# B&R Automation Studio project Soiled_PLC (part 15)

#### lpn.st - Implementation code
```iecst
(********************************************************************
 * COPYRIGHT --
 ********************************************************************
 * Program: pr
 * File: pr.st
 * Author: treamsbottom
 * Created: July 16, 2015
 ********************************************************************
 * Implementation of program pr
 ********************************************************************)
//V1.00.1 First Release
PROGRAM _INIT
//Configuration
mySeq						:= 31;	//Sequence number
myIO						:= 114;
myZone						:= 1;

myBag						:= 0; //Buffer Bag
myBuffBag					:= 0;

mySelectedLU_reg			:= mySeq; // D register to store selected loaded unit

bufferSettleTime			:= 300;

alarm						ACCESS ADR(Alarm[mySeq]);
bag							ACCESS ADR(Bag[myBag]);
//bag_buff					ACCESS ADR(Bag[myBuffBag]);

END_PROGRAM

PROGRAM _CYCLIC
//Inputs
i_bagAtBuffer				:= RequestRel.PN[1];//X[myIO].X01;

i_bagArriveLu[1]			:= X[myIO].X01;
i_bagArriveLu[2]			:= X[myIO].X02;

i_bagInRotaryPoint_front[1]	:= X[myIO].X03;
i_bagInRotaryPoint_rear[1]	:= X[myIO].X04;

i_bagInRotaryPoint_front[2]	:= X[myIO].X05;
i_bagInRotaryPoint_rear[2]	:= X[myIO].X06;

//Create the q for which loading unit to send to.
// N.B These input conditions are used to arrive the bag.
luWaitingLongest.input[1] := Request.LU[1]; //Loading unit does not have an empty bag space
luWaitingLongest.input[2] := NOT X[23].X01 AND NOT X[23].X02 AND NOT Y[23].Y05 AND NOT Y[23].Y06; //Loading unit 2 buffer.
luWaitingLongest.settleTime := 10;
luWaitingLongest();

o_openBuffer			:= FALSE;
o_straight				:= FALSE; // select all straight rails

FOR n := 0 TO MAX_LOADING_UNITS DO
	o_openFrontStop[n] 	:= FALSE;
	o_openRearStop[n] 	:= FALSE;
	o_rotate[n] 		:= FALSE;
END_FOR;

IF (myBag = 0) THEN
	alarm.Bag	:= mySeq + 10000;
ELSE
	alarm.Bag	:= myBag;
END_IF;

alarm.Name 		:= 0;
alarm.Beacon	:= TRUE;
alarm.Extra		:= 0;
alarm.Time		:= 3000;

//Setup Sequence
step := D[900 + mySeq];
//Setup Pulse contact
pls := (step <> lastStep);
lastStep := step;

//Sequence
IF (step = 0) THEN
	//Disabled
END_IF;

//Step 1 reset points & switch check
ton_10ms_reset(IN:=((step = 1) AND NOT Std.HaltSysZone[myZone]), PT:= 400);
IF (step = 1) THEN
	switchCheck := TRUE;
	FOR n := 1 TO MAX_LOADING_UNITS DO
		IF (i_bagArriveLu[n] OR i_bagInRotaryPoint_front[n] OR i_bagInRotaryPoint_rear[n]) THEN
			switchCheck := FALSE;
			EXIT;
		END_IF;
	END_FOR;

	o_straight := NOT Std.HaltSysZone[myZone];
	IF ton_10ms_reset.Q AND switchCheck THEN
		D[900 + mySeq] := 2;
		Count[mySeq] := Count[mySeq] + 1;
	ELSIF NOT switchCheck THEN
		alarm.Name := ALM_SWITCH_FAULT;
		alarm.Time := 0;
	END_IF;
END_IF;

ton_10ms_SettledBuffer(IN:= i_bagAtBuffer,PT:= bufferSettleTime);
//Wait for at bag buffer and  decide where to send bag
IF (step = 2) THEN
	 bagWaiting := (ton_10ms_SettledBuffer.Q AND ((bag.Cat > 0) OR(myBag = 0)));
	IF bagWaiting AND (luWaitingLongest.waitingLongest > 0)  AND NOT Std.HaltSysZone[myZone] THEN
		D[mySelectedLU_reg] := luWaitingLongest.waitingLongest; // Store the selected loaded unit to a D register so we won;t lose it
		D[900 + mySeq] := 3;
	END_IF;
	IF (myBag > 0) AND ton_10ms_SettledBuffer.Q  AND (bag.Cat = 0) THEN
		alarm.Name := ALM_BAG_DATA_ERROR;
	END_IF;
END_IF;

loadingUnit := D[mySelectedLU_reg];
//open buffer and wait for trolley past stop
releaseValid := (loadingUnit > 0);
IF (step = 3) THEN
	//o_straight := 1;
	o_openBuffer := releaseValid;
	FOR n := loadingUnit TO 1 BY -1 DO;
		o_openFrontStop[n] := 1;	// Open all front stops up to and including the selected unit;
		o_openRearStop[n-1] := 1;	// Open all rear stops up to the selected unitl
	END_FOR;
	IF i_bagInRotaryPoint_rear[loadingUnit] OR i_bagArriveLu[loadingUnit] THEN //i_bagArriveLu[loadingUnit]
		D[900 + mySeq] := 4;
	END_IF;
	IF releaseValid  AND NOT Std.HaltSysZone[myZone] THEN
		alarm.Name := ALM_BAG_NOT_ARRIVED;
	END_IF;
END_IF;

//bag settles in rotary points.
ton_SettledInPoint(IN:= (i_bagInRotaryPoint_front[loadingUnit] AND i_bagInRotaryPoint_rear[loadingUnit]), PT := 300);
IF (step = 4) THEN
	//o_straight := 1;
	FOR n := loadingUnit TO 1 BY -1 DO;
		o_openFrontStop[n-1] := 1;	// Open all rear stops up to the selected unitl
		o_openRearStop[n-1] := 1;	// Open all rear stops up to the selected unitl
	END_FOR;
	IF ton_SettledInPoint.Q   AND NOT Std.HaltSysZone[myZone] THEN
		D[900 + mySeq] := 5;
	ELSIF NOT Std.HaltSysZone[myZone] THEN
		alarm.Name := ALM_BAG_NOT_SETTLED;
	END_IF;
END_IF;

//rotate points
ton_rotatePoints(IN:= (step = 5),PT:= 400);
IF (step = 5) THEN
	o_rotate[loadingUnit] := 1;
	IF ton_rotatePoints.Q AND NOT Std.HaltSysZone[myZone] THEN
		D[900 + mySeq] := 6;
	END_IF;
END_IF;

//release bag
IF (step = 6) THEN
	o_rotate[loadingUnit] := 1;
	o_openFrontStop[loadingUnit] := luWaitingLongest.input[loadingUnit];
	o_openRearStop[loadingUnit] := luWaitingLongest.input[loadingUnit];
	IF NOT luWaitingLongest.input[loadingUnit] THEN
		D[900 + mySeq] := 1;
	END_IF;
	alarm.Name := ALM_BAG_NOT_RELEASED;
END_IF;

//-----------------------------------
//PLC Outputs - adjust TO suit system
//-----------------------------------

//Y[myIO].Y05 := o_openBuffer;
EnableRel.PN[1]		:= o_openBuffer;

Y[380].Y01	:= o_straight;
Y[380].Y02  := o_rotate[1];
Y[380].Y03	:= o_straight;
Y[380].Y04  := o_rotate[1];
Y[380].Y05  := o_openFrontStop[1];
Y[380].Y06  := o_openRearStop[1];

Y[382].Y01	:= o_straight;
Y[382].Y02  := o_rotate[2];
Y[382].Y03	:= o_straight;
Y[382].Y04  := o_rotate[2];
Y[382].Y05  := o_openFrontStop[2];
Y[382].Y06  := o_openRearStop[2];

//Alarms
timerAlarm(IN := NOT pls AND (alarm.Name > 0),PT:= alarm.Time);

alarm.On 	:= timerAlarm.Q;
alarm.ET 	:= timerAlarm.ET;

END_PROGRAM
```

#### lpn.var - Local variables
```iecst
(********************************************************************
 * COPYRIGHT --
 ********************************************************************
 * Program: pr
 * File: pr.var
 * Author: treamsbottom
 * Created: July 16, 2015
 ********************************************************************
 * Local variables of program pr
 ********************************************************************)
VAR CONSTANT
	MAX_LOADING_UNITS : USINT := 2;
END_VAR
VAR
	mySeq : UINT;
	myIO : UINT;
	myZone : UINT;
	myBag : UINT;
	i_bagAtBuffer : BOOL;
	o_openBuffer : BOOL;
	step : UINT;
	pls : BOOL;
	timerAlarm : TON_10ms;
END_VAR
VAR RETAIN
	lastStep : UINT;
END_VAR
VAR
	bufferSettleTime : UDINT;
	myOutBag : UINT;
	myBuffBag : UINT;
	myCan : UINT;
	alarm : REFERENCE TO Alm;
	bag : REFERENCE TO Bag_typ;
	bag_buff : REFERENCE TO Bag_typ;
	bag_out : REFERENCE TO Bag_typ;
	can : REFERENCE TO CAN_Vars;
	ton_10ms_reset : TON_10ms := (0);
	bagWaiting : BOOL := 0;
	ton_10ms_SettledBuffer : TON_10ms := (0);
	luWaitingLongest : getWaitingLongest := (0);
	mySelectedLU_reg : UINT := 0;
	loadingUnit : UINT := 0;
	releaseValid : BOOL := 0;
	o_openFrontStop : ARRAY[0..MAX_LOADING_UNITS] OF BOOL := [0];
	o_openRearStop : ARRAY[0..MAX_LOADING_UNITS] OF BOOL := [0];
	i_bagArriveLu : ARRAY[0..MAX_LOADING_UNITS] OF BOOL := [0];
	o_rotate : ARRAY[0..MAX_LOADING_UNITS] OF BOOL := [0];
	o_straight : BOOL := FALSE;
	i_bagInRotaryPoint_front : ARRAY[0..MAX_LOADING_UNITS] OF BOOL := [0];
	i_bagInRotaryPoint_rear : ARRAY[0..MAX_LOADING_UNITS] OF BOOL := [0];
	ton_SettledInPoint : TON_10ms := (0);
	ton_rotatePoints : TON_10ms := (0);
	switchCheck : BOOL := 0;
	n : UINT := 0;
END_VAR
```

### Program Logical/BaseStandards/TwinRailLoadingUnit/lpf (IEC, version 1.00.1) - *Twin rail loading offgoing

#### lpf.st - Implementation code
```iecst
(********************************************************************
 * COPYRIGHT --
 ********************************************************************
 * Program: pr
 * File: pr.st
 * Author: treamsbottom
 * Created: July 16, 2015
 ********************************************************************
 * Implementation of program pr
 ********************************************************************)
//V1.00.1 First Release
PROGRAM _INIT
//Configuration
mySeq						:= 32;	//Sequence number
myIO						:= 115;	// IO for switches
myZone						:= 1;
myPF						:= 1;

myBag						:= 207; //transit Bag
myRelLine					:= 0; // Release Line - Set to 0 to Request Release

myLuBag[1]					:= 203;
myLuBag[2]					:= 201;

mySelectedLU_reg			:= mySeq; // D register to store selected loaded unit
bufferSettleTime			:= 300;

myOutBag					:= Line[myRelLine].LastBag;

alarm						ACCESS ADR(Alarm[mySeq]);
bag							ACCESS ADR(Bag[myBag]);
bag_out						ACCESS ADR(Bag[myOutBag]);
line_release				ACCESS ADR(Line[myRelLine]);

END_PROGRAM

PROGRAM _CYCLIC
//Inputs

i_bagInRotaryPoint_front[1]	:= X[myIO].X03;
i_bagInRotaryPoint_rear[1]	:= X[myIO].X04;

i_bagInRotaryPoint_front[2]	:= X[myIO].X05;
i_bagInRotaryPoint_rear[2]	:= X[myIO].X06;

i_bagAtBufferOut 		:= FALSE; // Any Single bag buffer out IO.
i_bufferOutOpen			:= FALSE;

//Create the q for which loading unit to send to.
// N.B These input conditions are used to arrive the bag.
luWaitingLongest.input[1] := X[21].X03 AND X[21].X04 AND (Bag[myLuBag[1]].Cat > 0); //Loading unit does not have an full bag space
luWaitingLongest.input[2] := RequestRel.LU[2];
luWaitingLongest.settleTime := bufferSettleTime;
luWaitingLongest();

o_straight				:= FALSE; // select all straight rails
Request.PF[myPF]		:= FALSE;
RequestRel.PF[myPF]		:= FALSE;

FOR n := 0 TO MAX_LOADING_UNITS DO
	o_openStops[n]		:= FALSE;	// Stop on rotary points.
	o_rotate[n] 		:= FALSE;
	o_release[n]		:= FALSE;	// Release from loading unit or buffer.
END_FOR;

IF (myBag = 0) THEN
	alarm.Bag	:= mySeq + 10000;
ELSE
	alarm.Bag	:= myBag;
END_IF;

alarm.Name 		:= 0;
alarm.Beacon	:= TRUE;
alarm.Extra		:= 0;
alarm.Time		:= 3000;

//Setup Sequence
step := D[900 + mySeq];
//Setup Pulse contact
pls := (step <> lastStep);
lastStep := step;

//Sequence
IF (step = 0) THEN
	//Disabled
END_IF;

//Step 1 reset points & switch check
ton_10ms_reset(IN:=((step = 1) AND NOT Std.HaltSysZone[myZone]), PT:= 400);
IF (step = 1) THEN
	switchCheck := TRUE;
	FOR n := 1 TO MAX_LOADING_UNITS DO
		IF (i_bagInRotaryPoint_front[n] OR i_bagInRotaryPoint_rear[n]) THEN
			switchCheck := FALSE;
			EXIT;
		END_IF;
	END_FOR;
	o_straight := NOT Std.HaltSysZone[myZone];
	IF ton_10ms_reset.Q AND switchCheck AND (bag.Cat = 0) THEN
		D[900 + mySeq] := 2;
		Count[mySeq] := Count[mySeq] + 1;
	ELSIF NOT switchCheck THEN
		alarm.Name := ALM_SWITCH_FAULT;
		alarm.Time := 0;
	ELSIF (bag.Cat > 0) THEN
		alarm.Name := ALM_BAG_DATA_ERROR;
		alarm.Time := 0;
	END_IF;
END_IF;

//Wait for at bag buffer and  decide where to send bag
IF (step = 2) THEN
	releaseOk := (bag.Cat = 0);// We don;t have to check the loading unit bag data.. the queue is already checking it,
	IF releaseOk AND (luWaitingLongest.waitingLongest > 0)  AND NOT Std.HaltSysZone[myZone] THEN
		D[mySelectedLU_reg] := luWaitingLongest.waitingLongest; // Store the selected loaded unit to a D register so we won;t lose it
		D[900 + mySeq] := 3;
	ELSIF NOT releaseOk  AND NOT Std.HaltSysZone[myZone] THEN
		alarm.Name := ALM_BAG_DATA_ERROR;
		alarm.Time := 0;
	END_IF;
END_IF;

loadingUnit := D[mySelectedLU_reg];

//rotate points
ton_rotatePoints(IN:= ((step = 3) OR (step = 5)) ,PT:= 400);
IF (step = 3) THEN
	o_rotate[loadingUnit] := 1;
	IF ton_rotatePoints.Q  AND NOT Std.HaltSysZone[myZone] THEN
		D[900 + mySeq] := 4;
	END_IF;
END_IF;

releaseOk := (bag.Cat = 0) AND (Bag[myLuBag[loadingUnit]].Cat > 0) AND NOT Std.HaltSysZone[myZone];
//bag settles in point
ton_SettledInPoint(IN:= (i_bagInRotaryPoint_front[loadingUnit] AND i_bagInRotaryPoint_rear[loadingUnit]), PT := 300);
IF (step = 4) THEN
	o_rotate[loadingUnit] := 1;
	o_release[loadingUnit] := releaseOk;
	IF ton_SettledInPoint.Q AND releaseOk  THEN
		bag := Bag[myLuBag[loadingUnit]];
		Bag[myLuBag[loadingUnit]] := Bag[0];
		D[900 + mySeq] := 5;
	ELSIF NOT releaseOk AND NOT Std.HaltSysZone[myZone] THEN
		IF (bag.Cat > 0) THEN
			alarm.Name := ALM_BAG_DATA_ERROR;
			alarm.Time := 0;
		ELSE
			alarm.Name 	:= ALM_BAG_DATA_ERROR;
			alarm.Time 	:= 0;
			alarm.Bag 	:= myLuBag[loadingUnit];
		END_IF;
	ELSE
		alarm.Name := ALM_BAG_NOT_SETTLED;
	END_IF;
END_IF;

//rotate points back to straight
IF (step = 5) THEN
	o_straight	:= 1;
	IF ton_rotatePoints.Q AND NOT EnableRel.PF[myPF] THEN
		D[900 + mySeq] := 6;
	ELSIF EnableRel.PF[myPF] THEN
		alarm.Name := ALM_BAG_DATA_ERROR;
	END_IF;
END_IF;

//Check for line space.
IF (step = 6) THEN
	releaseValid := (NOT i_bagAtBufferOut AND NOT i_bufferOutOpen AND (bag.Cat > 0) AND (bag_out.Cat = 0));
	o_straight	:= 1;
	IF NOT Std.HaltSysZone[myZone] THEN
		IF (myRelLine > 0) THEN
			IF (line_release.Clear AND releaseValid) THEN
				C[myRelLine] := 0;
				D[900 + mySeq] := 7;
			END_IF;
			IF (line_release.Clear AND i_bagAtBufferOut) THEN
				alarm.Name := ALM_SWITCH_FAULT;
			ELSIF (bag.Cat = 0) THEN
				alarm.Name := ALM_BAG_DATA_ERROR;
				alarm.Time := 0;
			ELSIF line_release.Clear AND (bag_out.Cat > 0) THEN
				alarm.Name := ALM_BAG_DATA_ERROR;
				alarm.Bag := myOutBag;
				alarm.Time := 0;
			END_IF;
		ELSE
			RequestRel.PF[myPF] := releaseValid;
			IF EnableRel.PF[myPF] AND releaseValid THEN
				D[900 + mySeq] := 7;
			ELSIF (myBag > 0) AND (bag.Cat = 0) THEN
				alarm.Name := ALM_BAG_DATA_ERROR;
				alarm.Time := 0;
			ELSIF (myOutBag > 0) AND (bag_out.Cat > 0) THEN
				alarm.Name := ALM_BAG_DATA_ERROR;
				alarm.Bag := myOutBag;
				alarm.Time := 0;
			END_IF;
		END_IF;
	END_IF;
END_IF;

//Release bag.
IF (step = 7) THEN
	IF (NOT i_bagAtBufferOut AND NOT i_bufferOutOpen AND (bag.Cat > 0) AND (bag_out.Cat = 0) AND NOT Std.HaltSysZone[myZone]) THEN
		releaseValid := 1;
	END_IF;
	FOR n := loadingUnit TO 1 BY - 1 DO
		o_openStops[n] := releaseValid;
	END_FOR;
	o_straight := 1;
	IF releaseValid THEN
		IF (myRelLine > 0) THEN
			IF line_release.Trip THEN
				bag_out := bag;
				bag := Bag[0];
				D[900 + mySeq] := 1;
			END_IF;
		ELSE
			IF NOT EnableRel.PF[myPF] AND (bag.Cat = 0) THEN // Make sure data is copied out by enabling sequence.
				D[900 + mySeq] := 1;
			ELSIF NOT EnableRel.PF[myPF] AND (bag.Cat > 0) THEN
				alarm.Name := ALM_BAG_DATA_ERROR;
			END_IF;
		END_IF;
	ELSIF i_bagAtBufferOut OR i_bufferOutOpen THEN
		alarm.Name := ALM_SWITCH_FAULT;
		alarm.Time := 0;
	ELSIF (bag.Cat = 0) THEN
		alarm.Name := ALM_BAG_DATA_ERROR;
		alarm.Time := 0;
	ELSIF (bag_out.Cat > 0) THEN
		alarm.Name := ALM_BAG_DATA_ERROR;
		alarm.Bag := myOutBag;
		alarm.Time := 0;
	END_IF;
ELSE
	releaseValid := 0;
END_IF;

//-----------------------------------
//PLC Outputs - adjust TO suit system
//-----------------------------------

Y[21].Y07 := o_release[1];
Y[21].Y08 := o_release[1];

EnableRel.LU[2] := o_release[2];

Y[381].Y01	:= o_straight;
Y[381].Y02  := o_rotate[1];
Y[381].Y03	:= o_straight;
Y[381].Y04  := o_rotate[1];
Y[381].Y05  := o_openStops[1];
Y[381].Y06  := o_openStops[1];

Y[383].Y01	:= o_straight;
Y[383].Y02  := o_rotate[2];
Y[383].Y03	:= o_straight;
Y[383].Y04  := o_rotate[2];
Y[383].Y05  := o_openStops[2];
Y[383].Y06  := o_openStops[2];

//Alarms
timerAlarm(IN := NOT pls AND (alarm.Name > 0),PT:= alarm.Time);

alarm.On 	:= timerAlarm.Q;
alarm.ET 	:= timerAlarm.ET;

END_PROGRAM
```

#### lpf.var - Local variables
```iecst
(********************************************************************
 * COPYRIGHT --
 ********************************************************************
 * Program: pr
 * File: pr.var
 * Author: treamsbottom
 * Created: July 16, 2015
 ********************************************************************
 * Local variables of program pr
 ********************************************************************)
VAR CONSTANT
	MAX_LOADING_UNITS : USINT := 2;
END_VAR
VAR
	mySeq : UINT;
	myIO : UINT;
	myZone : UINT;
	myBag : UINT;
	step : UINT;
	pls : BOOL;
	timerAlarm : TON_10ms;
END_VAR
VAR RETAIN
	lastStep : UINT;
END_VAR
VAR
	myOutBag : UINT;
	myLuBag : ARRAY[0..MAX_LOADING_UNITS] OF UINT;
	alarm : REFERENCE TO Alm;
	bag : REFERENCE TO Bag_typ;
	bag_out : REFERENCE TO Bag_typ;
	ton_10ms_reset : TON_10ms := (0);
	luWaitingLongest : getWaitingLongest := (0);
	mySelectedLU_reg : UINT := 0;
	loadingUnit : UINT := 0;
	releaseValid : BOOL := 0;
	o_openStops : ARRAY[0..MAX_LOADING_UNITS] OF BOOL := [0];
	o_rotate : ARRAY[0..MAX_LOADING_UNITS] OF BOOL := [0];
	o_straight : BOOL := FALSE;
	i_bagInRotaryPoint_front : ARRAY[0..MAX_LOADING_UNITS] OF BOOL := [0];
	i_bagInRotaryPoint_rear : ARRAY[0..MAX_LOADING_UNITS] OF BOOL := [0];
	ton_SettledInPoint : TON_10ms := (0);
	ton_rotatePoints : TON_10ms := (0);
	switchCheck : BOOL := 0;
	o_release : ARRAY[0..MAX_LOADING_UNITS] OF BOOL := [0];
	releaseOk : BOOL := FALSE;
	myRelLine : UINT := 0;
	bufferSettleTime : UINT := 0;
	line_release : REFERENCE TO Line_Typ;
	i_bagAtBufferOut : BOOL := 0;
	i_bufferOutOpen : BOOL := 0;
	myPF : UINT := 0;
	n : UINT := 0;
END_VAR
```

### Program Logical/BaseStandards/11_spi1 (IEC) - * SPI1 Pneumatic Incline Up 1

#### 11_spi1.var
```iecst
VAR RETAIN
	STEP	:UINT;
	PLS	:BOOL;
	LASTSTEP	:UINT;
	BagSettled	:BOOL;
	BagSettledET	:TIME;
	O_OpenBufferStop	:BOOL;
	BagSettledBuffer	:BOOL;
	I_BaginIncline	:BOOL;
	BagSettledBufferET	:TIME;
	I_BagAtBuffer	:BOOL;
	I_CarrAtBottom	:BOOL;
	I_CarrAtTop	:BOOL;
	O_MoveDown	:BOOL;
END_VAR

VAR
	TempDownTime	:BOOL;
	TempDownTimeET	:TIME;
END_VAR
```

#### 11_spi1Cyclic.ab
```automation-basic
PROGRAM _CYCLIC
	(* cyclic program *)

;Sequence 11 - Pneumatic Incline 1 D[911]

;Incline Conveyor

;-----------------------------------------
;Revision 1.00 17/01/2006 D.J. First Issue
;-----------------------------------------

TON_10ms(O_MoveDown,1000,TempDownTime,TempDownTimeET)

I_BagAtBuffer			= X[8].X12
I_BaginIncline			= X[8].X13
I_CarrAtBottom			= X[8].X14
I_CarrAtTop				= X[8].X15

O_MoveDown 				= FALSE
O_OpenBufferStop		= FALSE

Request.PI[1]			= FALSE

Alarm[11].Name 			= 0
Alarm[11].Bag			= 10011
Alarm[11].Beacon		= TRUE

;Setup Sequence
;--------------
STEP = D[911]
;Setup Pulse contact
PLS = (STEP <> LASTSTEP)
LASTSTEP = STEP

;Allow carriage to go up to top
IF (STEP = 1) THEN
	IF I_CarrAtTop THEN
		D[911] = 2
	ENDIF
	IF NOT Std.HaltSys THEN
		Alarm[11].Name = almCarriageMoveFault
	ENDIF
ENDIF

;Check for bag at buffer
TON_10ms(I_BagAtBuffer,300,BagSettledBuffer,BagSettledBufferET)
IF (STEP = 2) THEN
	IF BagSettledBuffer THEN
		D[911] = 3
	ENDIF
ENDIF

;Open Buffer Stop on steps 3
IF (STEP >= 3) AND (STEP <= 3) THEN
	O_OpenBufferStop = TRUE
ENDIF

;Wait for bag in incline
IF (STEP = 3) THEN
	IF I_BaginIncline THEN
		D[911] = 4
	ENDIF
;	Alarm[11].Name = almBagNotArrived
ENDIF

;Let bag settle at base of incline
TON_10ms(I_BaginIncline,300,BagSettled,BagSettledET)
IF (STEP = 4) THEN
	IF BagSettled THEN
		D[911] = 5
	ENDIF
	Alarm[11].Name = almBagNotSettled
ENDIF

;Move carriage down to bottom
IF (STEP = 5) THEN
	O_MoveDown = TRUE
	IF I_CarrAtBottom THEN
		D[911] = 6
	ENDIF
	Alarm[11].Name = almCarriageMoveFault
ENDIF

;Allow carriage to move up to top
IF (STEP = 6) THEN
	IF I_CarrAtTop THEN
		D[911] 	= 7
	ENDIF
	Alarm[11].Name = almCarriageMoveFault
ENDIF

;Wait for space at empty bag buffer
IF (STEP = 7) THEN
	Request.PI[1] = TRUE
	IF Line[18].Clear AND BagSettled THEN
		D[911] 	= 8
	ENDIF
ENDIF

;Move carriage down to bottom
IF (STEP = 8) THEN
	O_MoveDown = TRUE
	IF I_CarrAtBottom THEN
		D[911] = 9
	ENDIF
	Alarm[11].Name = almCarriageMoveFault
ENDIF

;Allow carriage to move up releasing bag
IF (STEP = 9) THEN
	IF PLS THEN
		C[18] = 0
	ENDIF
	IF Line[18].Trip THEN
		D[911] = 1
	ENDIF
	Alarm[11].Name = almBagNotReleased
ENDIF

;Alarms
TON_10ms(NOT PLS AND (Alarm[11].Name > 0),3000,Alarm[11].On,Alarm[11].ET)

Y[8].Y12 = O_OpenBufferStop
Y[8].Y13 = O_MoveDown
END_PROGRAM
```

### Program Logical/BaseStandards/41_stnsa1 (IEC) - *Sorting Stations--

#### stnsa.ab
```automation-basic
PROGRAM _CYCLIC
(* cyclic program *)

;Honeycombe Sorting Station Control
;----------------------------------------------------
;Revision 1.00 10/01/2002 D.J. First Issue
;Revision 2.00 07/02/2005 D.J. Removed Stn Mix
;Revision 3.00 22/08/2006 D.J. Changed to timer array
;----------------------------------------------------

mySeq = 34
Bank = 1

;Timers
OpenTime  = 700
CloseTime = 500

ContinuousSort = FALSE;(D[994] = 0)

;Lamp Test from TrackView
IF (BIT_TST(D[998],0) = 1) THEN
	LampTest = TRUE

ELSE
	LampTest = FALSE
ENDIF

	LOOP x = 1 TO Ldg[Bank].NoStations DO
		n = Ldg[Bank].Stations[x]

		;Parts Loads
		TimerPartLoad[n].IN		= I_PartLoad[n]
		TimerPartLoad[n].PT		= 100
		TimerPartLoad[n] FUB TON_10ms()

		IF TimerPartLoad[n].Q THEN
			D[800 + n] = 1
		ENDIF

		;Bag open timers
		TimerOpen[n].IN 		= OpenBag[n]
		TimerOpen[n].PT			= OpenTime
		TimerOpen[n] FUB TON_10ms()

		BagOpened[n] 			= TimerOpen[n].Q
		BagOpenedET[n]			= TimerOpen[n].ET

		;Bag closed timers
		TimerClosed[n].IN 		= NOT OpenBag[n]
		TimerClosed[n].PT		= CloseTime
		TimerClosed[n] FUB TON_10ms()

		BagClosed[n] 			= TimerClosed[n].Q
		BagClosedET[n]			= TimerClosed[n].ET

		;Update bag weight
		StnBag = LDG_GetBagFromStation(Std.StationBagsStart,n)
		Bag[StnBag].Wgt 		= Stn[n].Weight
		Bag[StnBag].Cnt 		= Stn[n].Count

		;Update Bag ID if cleared or zero
		IF ((BidStn > 0) AND (Bag[StnBag].Bid = 0) AND (Bag[StnBag].Cat > 0)) THEN
			Bag[StnBag].Bid = UINT(BidStn)
			BidStn			= 0
		ENDIF

		;Move bags from Display buffer position into Search array,,
		myDisplayBag = LDG_GetBagFromStation(Std.StationBagDisplay,n)

		;Keep Weight Live on Display
		Bag[myDisplayBag].Wgt = Stn[n].Weight
		Update = FALSE
		IF (Bag[StnBag].Cat <> Bag[myDisplayBag].Cat) THEN
			Update = TRUE
		ELSE IF (Bag[StnBag].Cus <> Bag[myDisplayBag].Cus) THEN
			Update = TRUE
		ELSE IF (Bag[StnBag].Prg <> Bag[myDisplayBag].Prg) THEN
			Update = TRUE
		ENDIF
		IF (Bag[myDisplayBag].Cat = Std.MaxCats) THEN
			Update = FALSE ; Do not update bag if Empty Bag is assigned.
			CloseFlap[n] = TRUE
		ELSE
			CloseFlap[n] = FALSE
		ENDIF

		;Flap close after above SP2 for 1 second
		TimerFlapClose[n].IN 	= Stn[n].SP2 AND (Bag[myDisplayBag].Cat <> Std.MaxCats)
		TimerFlapClose[n].PT	= 200 ;4 sec
		TimerFlapClose[n] FUB TON_10ms()

		IF ContinuousSort THEN
			AutoPurgeTrig[n].CLK = Update
			AutoPurgeTrig[n] FUB R_TRIG()
			IF AutoPurgeTrig[n].Q THEN
				newBag[n] = TRUE
			ENDIF

			IF (newBag[n] AND Std.AutoPurge AND NOT Stn[n].CloseFlap AND NOT Stn[n].ManualRelease AND NOT Stn[n].Purge AND NOT Stn[n].PurgeReverse)THEN
				D[800 + n] = 2 ; Bag change detected automatically purge the station... Weight is check in ZZstn
				newBag[n] = FALSE
			ENDIF

			IF ((NOT Stn[n].CloseFlap AND NOT Stn[n].ManualRelease AND NOT Stn[n].Purge AND NOT Stn[n].PurgeReverse AND (D[800 + n] = 0)) OR  (Bag[StnBag].Cat = 0)) THEN ;AND NOT Stn[n].SP2 THEN
				IF Update THEN;(Update AND (n <> 12)) THEN
					myBid = Bag[StnBag].Bid
					Bag[StnBag] = Bag[myDisplayBag]
					Bag[StnBag].Bid = myBid
				ENDIF
			ENDIF
		ELSE
			IF Update THEN
				myBid = Bag[StnBag].Bid
				Bag[StnBag] = Bag[myDisplayBag]
				Bag[StnBag].Bid = myBid
			ENDIF
		ENDIF

		;Ensure Display Bag has a  Bag ID
		IF ((BidStn > 0) AND (Bag[myDisplayBag].Bid = 0) AND  (Bag[myDisplayBag].Cat > 0)) THEN
			Bag[myDisplayBag].Bid = UINT(BidStn)
			BidStn			= 0
		ENDIF

		Alarm[mySeq + n].Name 		= 0
		Alarm[mySeq + n].Bag		= StnBag
		Alarm[mySeq + n].Beacon	= FALSE
		Alarm[mySeq + n].Extra		= 0
		Alarm[mySeq + n].Time		= 4000

		Stn[n].LampOn 		= FALSE
		Stn[n].GreenLamp	= FALSE

		STEP = D[900 + mySeq + n]
		;Setup Pulse contact
		PLS[n] = (STEP <> LASTSTEP[n])
		LASTSTEP[n] = STEP

		;Step 0 - Disabled
		IF (STEP = 0) THEN
			Stn[n].LampOn = TRUE
			Stn[n].CloseFlap = ((Bag[StnBag].Cat <> Bag[myDisplayBag].Cat))
			Stn[n].QTime = 0
			Stn[n].ManualRelease = 0
			Stn[n].Purge = 0
			;Disabled
		ENDIF

		IF (STEP = 1) THEN
			Stn[n].LampOn = TRUE
			Stn[n].GreenLamp = FALSE
			Stn[n].CloseFlap = TRUE
			myStnReg = (n > 32)
			IF (myStnReg = 0)THEN
				myStnBit =	n - 1
			ELSE IF (myStnReg = 1)THEN
				myStnBit = 	n - 33
			ELSE
				myStnBit = 0
			ENDIF
			Std.PurgeBank[Bank].StationsStatus[myStnReg] = BIT_CLR(Std.PurgeBank[Bank].StationsStatus[myStnReg],myStnBit)

	;		Stn[n].Purge = FALSE
	;		Stn[n].PurgeReverse = FALSE
			IF D[900 + Std.StationBankReg + Bank] = n THEN
				D[900 + Std.StationBankReg + Bank] = 0
			ENDIF
			IF BagClosed[n] THEN
				D[900 + mySeq + n] = 2
			ENDIF
			Alarm[mySeq + n].Name = almStationNotClosed
		ENDIF

		IF (STEP = 2) THEN
			Stn[n].LampOn = ((Stn[n].SP1 AND Std.Clock2s) OR Stn[n].SP2 OR (Stn[n].SP3 AND Std.Clock200ms))
			Stn[n].GreenLamp = ((NOT Stn[n].SP2 AND NOT Stn[n].SP3) OR TimerFlapClose[n].Q)
			;Close the flaps when the bag is above SP2
			IF TimerFlapClose[n].Q OR Stn[n].ManualRelease OR Stn[n].Purge OR Stn[n].PurgeReverse THEN
				Stn[n].CloseFlap 	= ContinuousSort
			ENDIF
			;Stop flap closing / re-open is bag below 3kg
			IF (Stn[n].Weight < 30) THEN
				Stn[n].CloseFlap 	= FALSE
			ENDIF
			IF ((D[900 + Std.StationBankReg + Bank] = n) AND Ldg[Bank].EnableStnRelease) THEN
				D[900 + mySeq + n] = 3
			ENDIF
			IF ((Bag[StnBag].Prg > 0) AND Stn[n].SP3) THEN
				Alarm[mySeq + n].Name = almBagOverWeight
			ENDIF
		ENDIF

		IF (STEP = 3) THEN
			Stn[n].LampOn = TRUE
			Stn[n].CloseFlap = ContinuousSort
			Stn[n].GreenLamp = TimerFlapClose[n].Q

			AllowRelease[n]  = TRUE

			IF (BagOpened[n] AND ((Stn[n].Weight < 30) OR Test.Stations) AND Ldg[Bank].BeltHasRun) THEN
				Stn[n].QTime 	= 0
				D[900 + mySeq + n] = 1
			ENDIF
			IF (Stn[n].Weight >= 30) THEN
				Alarm[mySeq + n].Name = almStationNotEmpty
			ENDIF
		ELSE
			AllowRelease[n]= FALSE
		ENDIF

		OpenBag[n] = AllowRelease[n];(STEP = 3)

		;Lamp Test
		IF LampTest THEN
			Stn[n].LampOn = TRUE
		ENDIF

		;Alarm timer
		TimerAlarm[n].IN 	= NOT PLS[n] AND (Alarm[mySeq + n].Name > 0)
		TimerAlarm[n].PT	= Alarm[mySeq + n].Time
		TimerAlarm[n] FUB TON_10ms()

		Alarm[mySeq + n].ET	= TimerAlarm[n].ET
		Alarm[mySeq + n].On 	= TimerAlarm[n].Q

;	Y[300 + n].Y07 = Stn[n].LampOn
;	Y[300 + n].Y05 = Stn[n].CloseFlap OR testClose
;	Y[300 + n].Y06 = Stn[n].GreenLamp
;	Y[300 + n].Y04 = OpenBag[n]

ENDLOOP

;Outputs
;-------
;	YG05 = OpenBag[1]
;	YG06 = OpenBag[2]
;	YG07 = OpenBag[3]
;	YG08 = OpenBag[4]
;	YH05 = OpenBag[5]
;	YH06 = OpenBag[6]
;	YH07 = OpenBag[7]
;	YH08 = OpenBag[8]
;	YJ05 = OpenBag[9]
;	YJ06 = OpenBag[10]
;	YJ07 = OpenBag[11]
;	YJ08 = OpenBag[12]
;	YK05 = OpenBag[13]
;	YK06 = OpenBag[14]
;	YK07 = OpenBag[15]
;	YK08 = OpenBag[16]

	Y[31].Y05 = OpenBag[1] ;ok
	Y[31].Y06 = OpenBag[2]
	Y[31].Y07 = OpenBag[3]
	Y[31].Y08 = OpenBag[4]

	Y[32].Y05 = OpenBag[5];ok
	Y[32].Y06 = OpenBag[6]
	Y[32].Y07 = OpenBag[7]
	Y[32].Y08 = OpenBag[8]

	Y[33].Y05 = OpenBag[9]
	Y[33].Y06 = OpenBag[10]
	Y[33].Y07 = OpenBag[11]
	Y[33].Y08 = OpenBag[12]

	Y[34].Y05 = OpenBag[13]
	Y[34].Y06 = OpenBag[14]
	Y[34].Y07 = OpenBag[15]
	Y[34].Y08 = OpenBag[16]

	Y[31].Y01 = Stn[1].LampOn ;ok
	Y[31].Y02 = Stn[2].LampOn
	Y[31].Y03 = Stn[3].LampOn
	Y[31].Y04 = Stn[4].LampOn

	Y[32].Y01 = Stn[5].LampOn ;ok
	Y[32].Y02 = Stn[6].LampOn
	Y[32].Y03 = Stn[7].LampOn
	Y[32].Y04 = Stn[8].LampOn

	Y[33].Y01 = Stn[9].LampOn
	Y[33].Y02 = Stn[10].LampOn
	Y[33].Y03 = Stn[11].LampOn
	Y[33].Y04 = Stn[12].LampOn

	Y[34].Y01 = Stn[13].LampOn
	Y[34].Y02 = Stn[14].LampOn
	Y[34].Y03 = Stn[15].LampOn
	Y[34].Y04 = Stn[16].LampOn

END_PROGRAM
```

### Program Logical/BaseStandards/15_cdc1 (IEC) - * SDC2 Machine 2 CAN

#### 7_sdc2Cyclic.ab
```automation-basic
PROGRAM _CYCLIC
	(* cyclic program *)

;Sequence 7 - Discharger 2 D[907]

;-----------------------------------------
;Revision 1.00 19/12/2005 D.J. First Issue
;-----------------------------------------

DischargerEnable 		= ((D[13] > 0) AND NOT Std.HaltSys)

;I_BagAtBuffer			= X[6].X07
I_OpenBag				= CAN[2].DropLoad OR TestDrop
I_LoadDropped			= CAN[2].LoadDropped OR TestDropped
I_BagAtBuffer			= X[6].X06 OR TestBuffer
I_BagAtDischarger		= X[6].X08 OR TestAtDisch
I_BagEmpty			  	= TRUE

I_BagAtEmptyBuffer		= FALSE ;X[6].X13
O_EmptyBagBufferOpen	= FALSE ;Y[6].Y13

O_BagReady				= FALSE
O_OpenBuffer 			= FALSE
O_Steadys				= FALSE
O_Closer				= FALSE
O_OpenBag				= FALSE
O_OpenStop				= FALSE

Request.DC[2] 			= FALSE
Request.DCEmptyRelease[2] = FALSE
;Alarm
Alarm[7].Name 			= almNoAlarm ;Clear sequence alarm name
Alarm[7].Bag 			= 188
Alarm[7].Beacon			= TRUE
Alarm[7].Extra			= 0
Alarm[7].Time			= 3000

;Setup Sequence
STEP = D[907]
;Setup Pulse contact
PLS = (STEP <> LASTSTEP)
LASTSTEP = STEP

;Step 0 - Disabled
IF (STEP = 0) THEN
	;Disabled
ENDIF

;Check Status - Bag settled at buffer, no bag at discharger, bag at buffer on screen and no bag at discharger on the screen
TON_10ms(I_BagAtBuffer,300,SettledAtBuffer,SettledAtBufferET)
IF (STEP = 1) THEN
	IF (NOT I_BagAtDischarger AND  (Bag[188].Cat = 0) AND NOT Std.HaltSys AND DischargerEnable AND SettledAtBuffer) THEN
		Request.DC[2] = TRUE
		D[907] = 2
	ENDIF
	IF I_BagAtDischarger THEN
		;D[907] = 2
	ENDIF
	IF (Bag[188].Cat > 0) THEN
		Alarm[7].Name = almBagDataError
	ELSE IF I_BagAtDischarger THEN
		Alarm[7].Name = almSwitchFault
	ELSE IF (Bag[188].Cat > 0) AND NOT I_BagAtBuffer THEN
		Alarm[7].Name 	= almBagNotAtProx
		Alarm[7].Bag	= 188
	ELSE IF (Bag[188].Cat = 0) AND I_BagAtBuffer AND DischargerEnable  THEN
		Alarm[7].Name 	= almBagNotShownOnScreen
		Alarm[7].Bag	= 188
	ENDIF
ENDIF

;Wait for bag in discharger
IF (STEP = 2) THEN
	O_OpenBuffer 	= TRUE
	IF I_BagAtDischarger THEN
		D[907] = 3
	ENDIF
	Alarm[7].Name = almNoAlarm ;almBagNotArrived
ENDIF

;Let bag settle in discharger
TON_10ms(((STEP = 3) AND I_BagAtDischarger),1000,SettledAtDischarger,SettledAtDischargerET)
IF (STEP = 3) THEN
	IF (Bag[188].Cat = 0) AND (Bag[189].Cat > 0) THEN
		Bag[188] = Bag[189]
		Bag[189] = Bag[0]
	ENDIF
	IF SettledAtDischarger THEN
		D[907] = 4
	ENDIF
	Alarm[7].Name = almBagNotSettled
ENDIF

;Allow steadys to move down
TON_10ms((STEP = 4),400,SteadysDown,SteadysDownET)
IF (STEP = 4) THEN
	IF SteadysDown THEN
		D[907] = 5
	ENDIF
	IF (Bag[188].Cat = Std.MaxCats) THEN
		D[907] = 8
	ENDIF
ENDIF

;Steady cylinders on from steps 4 - 9
O_Steadys = ((STEP >= 4) AND (STEP <= 9))

;Bag opener on from step 5 - 8
O_OpenBag = ((STEP >= 6) AND (STEP <= 8))

CodeStep  = ((STEP >= 4) AND (STEP <= 5))

;Wash Codes
IF CodeStep THEN

	Weight = Bag[188].Wgt

	;round up weight to give to wash machine
	Remainder = SINT(Bag[188].Wgt MOD 10)
	IF (Remainder > 4) THEN
		WgtRound = (Weight + 10)
	ELSE
		WgtRound = Weight
	ENDIF

	;WashCodes
	;if Below the Machine limit of 99 and no WashCode has been entered then send the Category

	CAN[2].Category 	= Bag[188].Cat
	CAN[2].Customer 	= Bag[188].Cus
	CAN[2].Weight   	= (WgtRound / 10) ;rounded up weight divide by 10
	;CAN[1].DoubleLoad 	= (Batch > 0)
ELSE
	;CAN[2].Category 	= 0
	;CAN[2].Customer 	= 0
	;CAN[2].Weight   	= 0
	;CAN[1].DoubleLoad 	= FALSE

ENDIF

;Bag Ready to Washing Machine
IF (STEP = 5) THEN
	CAN[2].BagReady 		= TRUE

	IF I_OpenBag OR TestDischarger THEN
		D[907] = 6
	ENDIF
ELSE
	CAN[2].BagReady = FALSE
ENDIF

;Set LoadDropped to False
IF (STEP <> 6) THEN
	LoadDropped = FALSE
ENDIF

;Open Bag Until LoadDropped recieved and has been open for 6 seconds
TON_10ms((STEP = 6),600,MinOpen,MinOpenET) ;ET means Elapsed Time
TON_10ms((STEP = 6) AND NOT I_DischargerBagEmpty ,100,BagEmpty,BagEmptyET)

IF (STEP = 6) THEN

	;IF I_LoadDropped  OR TestDischarger THEN

		LoadDropped = TRUE
	;ENDIF

	IF (LoadDropped AND MinOpen) THEN
		;Write Report
		;------------

	ENDIF
	IF (LoadDropped AND MinOpen ) THEN
		IF (ReportUnloading[2].Cat = 0) THEN
			ReportUnloading[2].Cat = UINT(Bag[188].Cat)	;Category
			ReportUnloading[2].Cus = Bag[188].Cus		;Customer
			ReportUnloading[2].Wgt = Bag[188].Wgt		;Weight
			ReportUnloading[2].Cnt = 0					;Count
			ReportUnloading[2].Stn = 0					;Station
			ReportUnloading[2].Mcn = 2					;Machine
		ENDIF
		D[907] = 7
	ENDIF
	Alarm[7].Name = almLoadNotDropped
	ELSE
	LoadDropped = FALSE
ENDIF

;Change display to empty bag
IF (STEP = 7) THEN
	IF ((NOT I_OpenBag  AND I_BagEmpty) OR TestDrop) THEN
		Bag[188].Prg 	= Std.MaxProg
		Bag[188].Cat 	= Std.MaxCats
		Bag[188].Cus 	= Std.MaxCust

		D[907] 			= 8
	ENDIF
	Alarm[7].Name = almGeneralSequence
ENDIF

;Close bag
TON_10ms((STEP = 8),700,CloserDown,CloserDownET)
IF (STEP = 8) THEN
	O_Closer = TRUE
	IF CloserDown THEN
		D[907] = 9
	ENDIF
ENDIF

;Allow closer to go back up
TON_10ms((STEP = 9),700,CloserUp,CloserUpET)
IF (STEP = 9) THEN
	IF CloserUp THEN
		D[907] = 10
	ENDIF
ENDIF

;Allow steadys to go up
TON_10ms((STEP = 10),400,SteadyUp,SteadyUpET)
IF (STEP = 10) THEN
	IF SteadyUp THEN
		D[907] = 11
	ENDIF
ENDIF

;Request empty bag release
IF (STEP = 11) THEN
	Request.DCEmptyRelease[2] = TRUE
	IF Enable.DC[2] THEN
		;C[32]  = 0
		D[907] = 12
	ENDIF
ENDIF

;Open buffer stop - unitl bag out
IF (STEP = 12) THEN
	O_OpenStop = TRUE
	Bag[188].Cat = 0
	Bag[188].Cus = 0
	Bag[188].Wgt = 0
	IF NOT Enable.DC[2] THEN
		D[907] = 1
	ENDIF
	Alarm[7].Name = almBagNotReleased
ENDIF

;Alarms
TimerAlarm.IN 	= NOT PLS AND (Alarm[7].Name > 0)
TimerAlarm.PT 	= Alarm[7].Time
TimerAlarm FUB TON_10ms()
Alarm[7].On 	= TimerAlarm.Q
Alarm[7].ET 	= TimerAlarm.ET

;Outputs
Y[6].Y06 = O_OpenBuffer
Y[6].Y07 = O_Steadys
Y[6].Y08 = O_OpenBag
Y[6].Y09 = O_OpenStop
Y[6].Y10 = O_Closer
END_PROGRAM
```

### Program Logical/BaseStandards/zzcp10ser (IEC)

#### zzstnser.var
```iecst
VAR
	MixProgTyp : BOOL;
	BatchFound : BOOL;
	MixCusts : BOOL;
	MixProgs : BOOL;
	MatchCust : BOOL;
	MatchBags : BOOL;
	MatchProgType : BOOL;
	MatchProg : BOOL;
	MatchCat : BOOL;
	StartPurge : BOOL;
	MixCats : BOOL;
	BankValid : BOOL;
	LineValid : BOOL;
	BagInList : ARRAY[0..30] OF BOOL;
	StartPurgeET : UDINT;
	BagNum : UINT;
	BagWgt : UINT;
	Index : UINT;
	PurgeBagsQty : UINT;
	StnNum : UINT;
	BatchCount : UINT;
	s : UINT;
	BatchWeight : UINT;
	myBag : UINT;
	r : UINT;
	MaxReverseWeight : UINT;
END_VAR
VAR RETAIN
	LineSearchManual : UINT;
END_VAR
VAR
	NumberOfPurgeBags : UINT;
	x : UINT;
END_VAR
VAR RETAIN
	SearchLine : UINT;
END_VAR
VAR
	Bank : UINT;
	Choice : UINT;
	EndofBagArray : UINT;
	PurgeBatchSize : UINT;
	MaxBatchWieght : UINT;
END_VAR
VAR RETAIN
	n : UINT;
END_VAR
VAR
	t : UINT;
	myBag_x : UINT;
	myBag_n : UINT;
END_VAR
VAR RETAIN
	SearchFound : UINT;
END_VAR
VAR
	LineSearch : ARRAY[0..4] OF UINT;
	SearchBagArray : ARRAY[0..30] OF UINT;
	PurgeBags : ARRAY[0..30] OF UINT;
	PurgeBagsInWgtOrder : ARRAY[0..30] OF UINT;
	PurgeOn : UINT;
	StatusReg : ARRAY[0..1] OF UDINT;
	SearchIndex : USINT;
	ReSearch : BOOL;
	MisMatchedLoad : BOOL;
	y : INT;
	Break : BOOL;
	StnCat : UDINT;
	GetStn : UINT;
	TestTim : BOOL;
	myStartStop : UINT;
	b : UINT;
	TON_Purge : ARRAY[0..4] OF TON_10ms;
	myBatchWgt : UDINT;
	test : UDINT;
END_VAR
```

#### zzstnser.ab
```automation-basic
;-----------------------------------------------------
;Sorting Station Search Routine - No changes required!
;-----------------------------------------------------

;----------------------------------------
;Version 1.00 19/12/2005 First Issue D.J.
;Version 2.00 03/11/2010 Revised D.J.
;Version 3.00 19/07/2016 TR... Fix bug so multiple banks can release whilst purging..
;----------------------------------------

PROGRAM _CYCLIC

;Only one Bank / Loading VC can search in a given scan.

myStartStop			= 100 ; Start of Start Stops

IF myStartStop >= 100 THEN
	myStartStop = myStartStop + 7600
ENDIF

Bank = Bank + 1
IF (Bank > Std.MaxStationBanks) THEN
	Bank = 1
ENDIF
;Clear arrays
LOOP n = 0 TO Std.MaxWeighstations DO
	BagInList[n] = FALSE
	SearchBagArray[n] = 0
ENDLOOP

;Clear Array
LOOP b = 1 TO 4 DO
	Std.StnsToPurge[b] = FALSE
	LOOP n = 1 TO Ldg[b].NoStations DO
		x = Ldg[b].Stations[n]
		IF Stn[x].Purge THEN
			Std.StnsToPurge[b] = TRUE
		ENDIF
	ENDLOOP
	TON_Purge[b].IN = Std.StnsToPurge[b]
	TON_Purge[b].PT = 100
	TON_Purge[b] FUB TON_10ms()
	//TON_10ms(Std.StnsToPurge,100,StartPurge,StartPurgeET) ; use a timer to wait for all purge events to be recieved from trackview
ENDLOOP

MixCats			= (D[369] > 0)
MixCusts		= (D[366] > 0)	;Allow mixing of customers?
MixProgs		= (D[367] > 0)	;Allow mixing of Programs?
MixProgTyp		= (D[368] > 0) 	;Allow mixing of Program Types?

;Mix Options are enforced in Trackview - If we do it in the PLC we cannot turn off Mixing.
;IF MixProgTyp THEN
;	D[367] = 1 //Mix Progs
;	D[369] = 1 //Mix Cats
;ELSE IF MixProgs THEN					;IF mixing programs then category must be mixed also.....
;	D[369] =  1 // Mix Cats
;ENDIF

;IF Std.ReversingBelt THEN
	MaxReverseWeight	= D[370]			;Max weight to reverse..
;ELSE
;	MaxReverseWeight = 0
;ENDIF
;Send Status to Trackview -- BitWise OR to look at all banks

PurgeOn = (Std.PurgeBank[1].PurgeOn OR Std.PurgeBank[2].PurgeOn OR Std.PurgeBank[3].PurgeOn OR Std.PurgeBank[4].PurgeOn)
StatusReg[0] = (Std.PurgeBank[1].StationsStatus[0] OR Std.PurgeBank[2].StationsStatus[0] OR Std.PurgeBank[3].StationsStatus[0] OR Std.PurgeBank[4].StationsStatus[0])
StatusReg[1] = (Std.PurgeBank[1].StationsStatus[1] OR Std.PurgeBank[2].StationsStatus[1] OR Std.PurgeBank[3].StationsStatus[1] OR Std.PurgeBank[4].StationsStatus[1])
D[360] = PurgeOn
memcpy(ADR(D[371]),ADR(StatusReg),4)
;Used by other sequences that need to check for Line[x].SpaceBIT direct
;eg. Loading VC will look for Enable.Search = 3
Enable.Search = Bank

IF (Bank <= Std.MaxStationBanks) THEN

	IF (Ldg[Bank].Search = 1) THEN
		StartPurge = TON_Purge[Bank].Q
		Ldg[Bank].Found = 0
		Ldg[Bank].Line  = 0

		SearchFound = 0
		SearchLine  = 0

		Stn[0].QTime = 0

		LOOP x = 1 TO Ldg[Bank].NoStations DO
			n = Ldg[Bank].Stations[x]
			IF (Std.StnsToPurge[Bank] AND Std.AutoPurge) THEN	;Search through purge Stations to find bags that can be mixed

				IF Bank = 1 THEN
					Break
;					IF NOT TestTim THEN
;						GOTO Debug
;					ENDIF
				ELSE IF Bank = 2 THEN
					Break
				ENDIF
				;Purge doesn;t need to be in x loop so exit if > 1
				EXITIF x > 1
				IF StartPurge THEN
					PurgeBatchSize	= 0
					BatchFound = FALSE
					; 1st put all bags to be searched into an array to reduce scanning through all stations bags
					//LOOP r = 0 TO Std.MaxWeighstations DO
					LOOP r = 1 TO Ldg[Bank].NoStations DO
						Std.PurgeBank[Bank].PurgeBatch[r] = 0
						n = Ldg[Bank].Stations[r]
						IF Stn[n].Purge AND (Stn[n].Weight > 0) AND NOT BagInList[n] THEN //AND (r >= Ldg[Bank].StartStn) AND (r <= Ldg[Bank].EndStn)  THEN
							SearchBagArray[Ldg[Bank].NoStations] = LDG_GetBagFromStation(Std.StationBagsStart,n)
							BagInList[n] = TRUE
						ENDIF
						;Shuffle array
						LOOP s = Ldg[Bank].NoStations DOWNTO 1 DO
							IF (SearchBagArray[s-1] = 0) AND (SearchBagArray[s] > 0) THEN
								SearchBagArray[s-1] = SearchBagArray[s]
								SearchBagArray[s] = 0
								EndofBagArray = (s - 1)
							ENDIF
						ENDLOOP
					ENDLOOP
					;LOOP r = 0 TO EndofBagArray DO ; Start Searching through bags
					r = 0 ;Only search through from 1st bag in array as we already know it is to purge
					ReSearch = FALSE
					MisMatchedLoad = FALSE
					SearchIndex = 0
					StartSearch: ;Marker to re-search
					IF ReSearch THEN
						r = SearchIndex
					ENDIF
					LOOP s = 0 TO Std.MaxWeighstations DO
						PurgeBags[s] = 0
					ENDLOOP
					LOOP s = EndofBagArray DOWNTO 0 DO
						myBag_n = SearchBagArray[r]
						myBag_x = SearchBagArray[s]
						MatchCust = FALSE
						MatchCat = FALSE
						MatchProgType = FALSE
						MatchProg = FALSE
						BankValid = TRUE;((myBag_n >= Ldg[Bank].StartStn) AND (myBag_n <= Ldg[Bank].EndStn) AND (myBag_x >= Ldg[Bank].StartStn) AND (myBag_x <= Ldg[0].EndStn))

						;Check customer 1st
						IF (Bag[myBag_n].Cus = Bag[myBag_x].Cus) OR MixCusts THEN
							MatchCust = TRUE
						ENDIF
						IF (Bag[myBag_n].Cat = Bag[myBag_x].Cat) OR MixCats THEN
							MatchCat = TRUE
						ENDIF
						IF (Bag[myBag_n].Prg = Bag[myBag_x].Prg) OR MixProgs THEN
							MatchProg = TRUE
						ENDIF
						IF (D[2900 + Bag[myBag_n].Prg] = D[2900 + Bag[myBag_x].Prg]) OR MixProgTyp THEN
							MatchProgType = TRUE
						ENDIF

						MatchBags = (MatchCust AND MatchCat AND MatchProg AND MatchProgType AND BankValid)
						IF MatchBags THEN ; Put bag into another array so they can be best matched by weight
							;PurgeBags[0] = myBag_n
							PurgeBags[Std.MaxWeighstations] = myBag_x
							LOOP t = Std.MaxWeighstations DOWNTO 1 DO
								IF (PurgeBags[t] > 0) AND (PurgeBags[t-1] = 0) THEN
									PurgeBags[t -1] = PurgeBags[t]
									PurgeBags[t] = 0
									PurgeBatchSize	= t
								ENDIF
							ENDLOOP
						ENDIF
					ENDLOOP ; Ony research if no matching bags, and the bag searched is to small for a batch
					//Get Total weight of batch to see if matched bags meet minumum weight criteria.
					myBatchWgt = 0
					LOOP t = 0 TO PurgeBatchSize DO
						myBatchWgt = myBatchWgt + Bag[PurgeBags[t]].Wgt
					ENDLOOP
					//IF ((PurgeBatchSize = 1) AND (Bag[PurgeBags[0]].Wgt < MaxReverseWeight)) THEN
					IF ((PurgeBatchSize >= 1) AND (myBatchWgt < MaxReverseWeight)) THEN
						ReSearch = TRUE
						INC SearchIndex
						;Check when all bags have been searched...
						IF (SearchBagArray[SearchIndex] = 0) THEN
							;INC SearchIndex
							;The only bags left cannot be put in the same bag and should be classified as a mixed load.
							MisMatchedLoad = (SearchIndex > 1)
							LOOP y = 0 TO SearchIndex - 1 DO
								PurgeBags[y] = 	SearchBagArray[y]
							ENDLOOP
							PurgeBatchSize = SearchIndex
						ELSE
							GOTO StartSearch
						ENDIF
					ENDIF

					;ENDLOOP
					;Matching bags are in the array Purge Bags. Try to fit into a load?
					;Bag 0 in the array is that master.. This is the data that will go into a bag.. so we will get the batch weight from this program code.
					;Put all bag into wieght order highest first..
					LOOP r = 0 TO 30 DO
						BagInList[r] = FALSE
						PurgeBagsInWgtOrder[r] = 0
					ENDLOOP

					IF (PurgeBatchSize > 0) THEN
						//Find the lowest SP3 from all bag in the purge array...
						MaxBatchWieght = 0
						LOOP r = 0 TO ((SIZEOF(PurgeBags)/SIZEOF(PurgeBags[0])) - 1) DO
							EXITIF PurgeBags[r] = 0
							GetStn =  (PurgeBags[r] - Std.StationBagsStart + 1)
							IF (GetStn <= Std.MaxWeighstations) AND (D[4900 + GetStn] > 0) AND ((MaxBatchWieght > D[4900 + GetStn]) OR (MaxBatchWieght = 0))    THEN
								MaxBatchWieght = D[4900 + GetStn] ;SP3
							ENDIF
						ENDLOOP

						IF (MaxBatchWieght = 0) OR (MaxBatchWieght <= MaxReverseWeight) THEN
							 MaxBatchWieght = MaxReverseWeight + 100
						ENDIF

						LOOP r = 0 TO (PurgeBatchSize - 1) DO
							BagWgt = 0
							LOOP s = 0 TO (PurgeBatchSize - 1) DO
								IF (Bag[PurgeBags[s]].Wgt > 0) AND (Bag[PurgeBags[s]].Wgt > BagWgt) AND NOT BagInList[s] THEN
									BagWgt = Bag[PurgeBags[s]].Wgt
									BagNum = PurgeBags[s]
									Index = s
								ENDIF
							ENDLOOP
							PurgeBagsInWgtOrder[r] = BagNum
							BagInList[Index] = TRUE
						ENDLOOP ;
						IF (MaxBatchWieght > MaxReverseWeight) AND (Bag[PurgeBagsInWgtOrder[0]].Wgt > 0)THEN ; Check no errors in batch sizes.. Reverse all loads if fault
							;Now bags are in weight order make the best by adding the highest values until bag is full
							BatchWeight = 0
							PurgeBagsQty = 0
							;IF (Bag[PurgeBagsInWgtOrder[0]].Wgt  < MaxBatchWieght) THEN
							BatchWeight = Bag[PurgeBagsInWgtOrder[0]].Wgt
							BatchCount = Bag[PurgeBagsInWgtOrder[0]].Cnt
							Std.PurgeBank[Bank].PurgeBatch[0] = PurgeBagsInWgtOrder[0]
							;ENDIF
							LOOP r = 1 TO PurgeBatchSize DO ; Start from 1 as index 0 is highest weight so always in the array
								myBag = PurgeBagsInWgtOrder[r]
								IF ((Bag[myBag].Wgt + BatchWeight) <= MaxBatchWieght) THEN
									BatchWeight = Bag[myBag].Wgt + BatchWeight
									BatchCount = Bag[myBag].Cnt + BatchCount
									Std.PurgeBank[Bank].PurgeBatch[PurgeBatchSize] = myBag
									PurgeBagsQty = PurgeBagsQty + 1
								ENDIF
								;Shuffle down array
								LOOP s = PurgeBatchSize DOWNTO 1 DO
									IF (Std.PurgeBank[Bank].PurgeBatch[s] > 0) AND (Std.PurgeBank[Bank].PurgeBatch[s - 1] = 0) THEN
										Std.PurgeBank[Bank].PurgeBatch[s - 1] = Std.PurgeBank[Bank].PurgeBatch[s]
										Std.PurgeBank[Bank].PurgeBatch[s] = 0
									ENDIF
								ENDLOOP
								IF (r = PurgeBatchSize) AND (Std.PurgeBank[Bank].PurgeBatch[0] > 0) THEN
									BatchFound = TRUE
								ENDIF
							EXITIF BatchFound = TRUE
							ENDLOOP
						ENDIF
;					ELSE
;						GOTO ExitPurge ;Invalid purge..
					ENDIF
					IF BatchFound AND NOT MisMatchedLoad THEN ;Bags found;
						IF (BatchWeight >=  MaxReverseWeight) THEN ; Wieght it OK purge into Bag search for destination.

							IF Std.AutoLineAllocation THEN
								SearchFound  		= 99
								SearchLine   		= 0;LineSearch[Choice]
								Ldg[Bank].Search   	= 2
							ELSE	;
								;Check line choice 1st to 4th in order if any valid then exit loop
								;StnNum = (Std.PurgeBank[Bank].PurgeBatch[0] - (Std.StationBagsStart[Bank] - Ldg[Bank].StartStn)) ; Get station number from Bag number.
								StnCat =  Bag[Std.PurgeBank[Bank].PurgeBatch[0]].Prg

								LineSearch[1]   = D[3000 + StnCat]
								LineSearch[2]   = D[3100 + StnCat]
								LineSearch[3]   = D[3200 + StnCat]
								LineSearch[4]   = D[3300 + StnCat]

								LOOP Choice = 1 TO 4 DO
									LineValid = (D[myStartStop + LineSearch[Choice]] > 0)
									IF (LineSearch[Choice] > 0) AND (Line[LineSearch[Choice]].SpaceBIT >= 1) AND LineValid THEN
										SearchFound  		= 99
										SearchLine   		= LineSearch[Choice]
										Ldg[Bank].Search   	= 2
									ENDIF
									EXITIF (SearchFound > 0)
								ENDLOOP
							ENDIF
						ELSE ; Load/s is to small reverse.

							SearchFound  		= 98
							SearchLine   		= 0
							Ldg[Bank].Search   	= 2
						ENDIF
					ELSE IF MisMatchedLoad THEN
						SearchFound  		= 97
						SearchLine   		= 0
						Ldg[Bank].Search   	= 2
					ENDIF
					IF SearchFound > 90 THEN ;If bags are found remove from purging Q
						Std.PurgeBank[Bank].PurgeBagQty	= PurgeBagsQty

						Std.PurgeBank[Bank].PurgeBatchWieght = BatchWeight
						Std.PurgeBank[Bank].PurgeBatchCount	= BatchCount
;						LOOP r = 0 TO PurgeBagsQty - 1 DO
;							IF (Std.PurgeBank[Bank].PurgeBatch[r] > 0) THEN
;								StnNum = (Std.PurgeBank[Bank].PurgeBatch[r] - (Std.StationBagsStart[Bank] - Ldg[Bank].StartStn))
;								;Stn[StnNum].QTime = 0
;								;Stn[StnNum].Purge = FALSE
;							ENDIF
;						ENDLOOP
					ENDIF
				ENDIF
			ELSE IF ((Stn[n].QTime > 10) AND (Stn[n].QTime > Stn[0].QTime)) THEN

				;Destination has been given to bag by operator check
				LineSearchManual = Stn[n].DestManual

				IF Std.AutoLineAllocation THEN

					;Automatic Line Allocation - Line Space is never checked even if a destiantion has been edited
					SearchFound  		= n
					SearchLine   		= LineSearchManual
					Stn[0].QTime 		= Stn[n].QTime
					Ldg[Bank].Search   	= 2

				ELSE
					;1st 2nd 3rd and 4th Line choices
					LineSearch[1]   = D[4000 + n]
					LineSearch[2]   = D[4100 + n]
					LineSearch[3]   = D[4200 + n]
					LineSearch[4]   = D[4300 + n]

					;Always Search for at least 1 space
					IF (Stn[n].SpacesRequired = 0) THEN
						Stn[n].SpacesRequired = 1
					ENDIF

					;When manual is selected then the 1st 2nd 3rd and 4th are not checked
					IF (LineSearchManual > 0) THEN
						IF (Line[LineSearchManual].SpaceBIT > 0) THEN
							SearchFound  		= n
							SearchLine   		= LineSearchManual
							Stn[0].QTime 		= Stn[n].QTime
							Ldg[Bank].Search   	= 2
						ENDIF
					ELSE
							;Check line choice 1st to 4th in order if any valid then exit loop

						LOOP Choice = 1 TO 4 DO
							;Choice = 1
							LineValid = (D[myStartStop + LineSearch[Choice]] > 0)
							IF (LineSearch[Choice] > 0) AND (LineSearch[Choice] < 7) AND (Line[LineSearch[Choice]].SpaceBIT >= Stn[n].SpacesRequired) AND LineValid THEN
								SearchFound  		= n
								SearchLine   		= LineSearch[Choice]
								Stn[0].QTime 		= Stn[n].QTime
								Ldg[Bank].Search   	= 2

							ENDIF
							EXITIF (SearchFound > 0)

							IF (LineSearch[Choice] > 13) THEN
								IF (Line[9].SpaceBIT > 0) THEN
									SearchFound  		= n
									SearchLine   		= LineSearch[Choice]
									Stn[0].QTime 		= Stn[n].QTime
									Ldg[Bank].Search   	= 2
								ENDIF
							ENDIF

						ENDLOOP

					ENDIF

				ENDIF ;/AutoLineAllocation

			ENDIF

		ENDLOOP

		ExitPurge:
		IF (Ldg[Bank].Search = 2) THEN
			Ldg[Bank].Found  = SearchFound
			Ldg[Bank].Line   = SearchLine
		ELSE
			Ldg[Bank].Search = 0 ;Failed
		ENDIF

	ENDIF
ENDIF
Debug:

END_PROGRAM
```

### OPCuA.var
```iecst
(*OPCUa Tag Vars*)
VAR
	OPCuA_Display : ARRAY[0..MAX_DISPLAYS] OF OPCuA_Display_typ;
	OPCuA_Bag : ARRAY[0..MAX_BAGS] OF EncodedBag_typ;
END_VAR
```

### Program Logical/OPCuA/TestValues (IEC)

#### Variables.var
```iecst
VAR
	ton_Change : TON_10ms;
	n : INT;
	ChangeIndex : USINT;
END_VAR
```

#### Cyclic.st
```iecst
PROGRAM _CYCLIC

ton_Change.IN := NOT ton_Change.Q;
ton_Change.PT := 1000;
ton_Change();

Bag[221].Ur1 := 16#FF00;

FOR n := 221 TO 228 DO
	IF Bag[n].Wgt < 850 THEN
		Bag[n].Wgt := Bag[n].Wgt + 10;
	ELSE
		Bag[n].Wgt := 0;
	END_IF;
	IF ton_Change.Q THEN
		ChangeIndex := ChangeIndex + 1;
		CASE ChangeIndex OF
			1:
				IF Bag[n].Cat < 10 THEN
					Bag[n].Cat := Bag[n].Cat + 1;
				ELSE
					Bag[n].Cat := 0;
				END_IF;
				Bag[n].Prg := UDINT_TO_USINT(Bag[n].Cat);
			2:
				IF Bag[n].Cus < 10 THEN
					Bag[n].Cus := Bag[n].Cus + 1;
				ELSE
					Bag[n].Cus := 0;
				END_IF;
			ELSE
				ChangeIndex := 1;

		END_CASE;

	END_IF;
END_FOR;

END_PROGRAM
```

### Program Logical/OPCuA/OPCuA_Test (IEC)

#### Variables.var
```iecst
VAR CONSTANT
	CONSTANT_DISPLAY_01 : INT := 1;
	CONSTANT_DISPLAY_00 : INT := 0;
	CONSTANT_DISPLAY_02 : INT := 2;
END_VAR
```

#### Cyclic.st
```iecst
PROGRAM _CYCLIC

//DISPLAY 0 *****************************************************************************

	OPCuA_Display[CONSTANT_DISPLAY_00].Layout[0].backcolour := 16#BADA55;
	OPCuA_Display[CONSTANT_DISPLAY_00].Layout[1].backcolour := 16#BADA55;
	OPCuA_Display[CONSTANT_DISPLAY_00].Layout[2].backcolour := 16#BADA55;

	OPCuA_Display[CONSTANT_DISPLAY_00].Layout[0].displayID := '0';
	OPCuA_Display[CONSTANT_DISPLAY_00].Layout[1].displayID := '1';
	OPCuA_Display[CONSTANT_DISPLAY_00].Layout[2].displayID := '2';

	OPCuA_Display[CONSTANT_DISPLAY_00].Layout[0].wgt     := OPCuA_Display[CONSTANT_DISPLAY_00].Layout[0].wgt + 10;
	OPCuA_Display[CONSTANT_DISPLAY_00].Layout[1].wgt     := OPCuA_Display[CONSTANT_DISPLAY_00].Layout[1].wgt + 10;
	OPCuA_Display[CONSTANT_DISPLAY_00].Layout[2].wgt     := OPCuA_Display[CONSTANT_DISPLAY_00].Layout[2].wgt + 10;

	//Layout 00
	IF OPCuA_Display[CONSTANT_DISPLAY_00].Layout[0].wgt > 900 THEN
		OPCuA_Display[CONSTANT_DISPLAY_00].Layout[0].wgt := 0;
	END_IF

	// Layput 01
	IF OPCuA_Display[CONSTANT_DISPLAY_00].Layout[1].wgt > 900 THEN
		OPCuA_Display[CONSTANT_DISPLAY_00].Layout[1].wgt := 0;
	END_IF

	IF OPCuA_Display[CONSTANT_DISPLAY_00].Layout[1].wgt > 400 THEN
		OPCuA_Display[CONSTANT_DISPLAY_00].Layout[1].displayID := '0';
		OPCuA_Display[CONSTANT_DISPLAY_00].Layout[1].cus := 3;
		OPCuA_Display[CONSTANT_DISPLAY_00].Layout[1].prg := 1;
		OPCuA_Display[CONSTANT_DISPLAY_00].Layout[1].cat := 1;
	END_IF

	IF OPCuA_Display[CONSTANT_DISPLAY_00].Layout[1].wgt > 800 THEN
		OPCuA_Display[CONSTANT_DISPLAY_00].Layout[1].cus := 2;
		OPCuA_Display[CONSTANT_DISPLAY_00].Layout[1].prg := 2;
		OPCuA_Display[CONSTANT_DISPLAY_00].Layout[1].cat := 2;
	END_IF

	// Layout 03
	IF OPCuA_Display[CONSTANT_DISPLAY_00].Layout[2].wgt > 900 THEN
		OPCuA_Display[CONSTANT_DISPLAY_00].Layout[2].wgt := 0;
	END_IF

// DISPLAY 1 *****************************************************************************
	OPCuA_Display[CONSTANT_DISPLAY_01].Layout[0].backcolour := 16#BADA55;
	OPCuA_Display[CONSTANT_DISPLAY_01].Layout[1].backcolour := 16#BADA55;
	OPCuA_Display[CONSTANT_DISPLAY_01].Layout[2].backcolour := 16#BADA55;
	OPCuA_Display[CONSTANT_DISPLAY_01].Layout[3].backcolour := 16#BADA55;
	OPCuA_Display[CONSTANT_DISPLAY_01].Layout[4].backcolour := 16#BADA55;

	OPCuA_Display[CONSTANT_DISPLAY_01].Layout[0].displayID := '0';
	OPCuA_Display[CONSTANT_DISPLAY_01].Layout[1].displayID := '1';
	OPCuA_Display[CONSTANT_DISPLAY_01].Layout[2].displayID := '2';
	OPCuA_Display[CONSTANT_DISPLAY_01].Layout[3].displayID := '3';
	OPCuA_Display[CONSTANT_DISPLAY_01].Layout[4].displayID := '4';

	OPCuA_Display[CONSTANT_DISPLAY_01].Layout[0].wgt     := OPCuA_Display[CONSTANT_DISPLAY_01].Layout[0].wgt + 10;
	OPCuA_Display[CONSTANT_DISPLAY_01].Layout[1].wgt     := OPCuA_Display[CONSTANT_DISPLAY_01].Layout[1].wgt + 11;
	OPCuA_Display[CONSTANT_DISPLAY_01].Layout[2].wgt     := OPCuA_Display[CONSTANT_DISPLAY_01].Layout[2].wgt + 12;
	OPCuA_Display[CONSTANT_DISPLAY_01].Layout[3].wgt     := OPCuA_Display[CONSTANT_DISPLAY_01].Layout[3].wgt + 13;
	OPCuA_Display[CONSTANT_DISPLAY_01].Layout[4].wgt     := OPCuA_Display[CONSTANT_DISPLAY_01].Layout[4].wgt + 14;

	//LAYOUT 01
	IF OPCuA_Display[CONSTANT_DISPLAY_01].Layout[1].wgt > 900 THEN
		OPCuA_Display[CONSTANT_DISPLAY_01].Layout[1].wgt := 0;
	END_IF

	IF OPCuA_Display[CONSTANT_DISPLAY_01].Layout[1].wgt > 400 THEN
		OPCuA_Display[CONSTANT_DISPLAY_01].Layout[1].displayID := '0';
		OPCuA_Display[CONSTANT_DISPLAY_01].Layout[1].cus := 1;
		OPCuA_Display[CONSTANT_DISPLAY_01].Layout[1].prg := 1;
		OPCuA_Display[CONSTANT_DISPLAY_01].Layout[1].cat := 1;
	END_IF

	IF OPCuA_Display[CONSTANT_DISPLAY_01].Layout[1].wgt > 800 THEN
		OPCuA_Display[CONSTANT_DISPLAY_01].Layout[1].cus := 2;
		OPCuA_Display[CONSTANT_DISPLAY_01].Layout[1].prg := 2;
		OPCuA_Display[CONSTANT_DISPLAY_01].Layout[1].cat := 2;
	END_IF

	//LAYOUT 02
	IF OPCuA_Display[CONSTANT_DISPLAY_01].Layout[2].wgt > 900 THEN
		OPCuA_Display[CONSTANT_DISPLAY_01].Layout[2].wgt := 0;
	END_IF

	IF OPCuA_Display[CONSTANT_DISPLAY_01].Layout[2].wgt > 400 THEN
		OPCuA_Display[CONSTANT_DISPLAY_01].Layout[2].displayID := '0';
		OPCuA_Display[CONSTANT_DISPLAY_01].Layout[2].cus := 2;
		OPCuA_Display[CONSTANT_DISPLAY_01].Layout[2].prg := 2;
		OPCuA_Display[CONSTANT_DISPLAY_01].Layout[2].cat := 2;
	END_IF

	IF OPCuA_Display[CONSTANT_DISPLAY_01].Layout[2].wgt > 800 THEN
		OPCuA_Display[CONSTANT_DISPLAY_01].Layout[2].cus := 1;
		OPCuA_Display[CONSTANT_DISPLAY_01].Layout[2].prg := 1;
		OPCuA_Display[CONSTANT_DISPLAY_01].Layout[2].cat := 1;
	END_IF

	//LAYOUT 03
	IF OPCuA_Display[CONSTANT_DISPLAY_01].Layout[3].wgt > 900 THEN
		OPCuA_Display[CONSTANT_DISPLAY_01].Layout[3].wgt := 0;
	END_IF

	IF OPCuA_Display[CONSTANT_DISPLAY_01].Layout[3].wgt > 400 THEN
		OPCuA_Display[CONSTANT_DISPLAY_01].Layout[3].displayID := '0';
		OPCuA_Display[CONSTANT_DISPLAY_01].Layout[3].cus := 1;
		OPCuA_Display[CONSTANT_DISPLAY_01].Layout[3].prg := 1;
		OPCuA_Display[CONSTANT_DISPLAY_01].Layout[3].cat := 1;
	END_IF

	IF OPCuA_Display[CONSTANT_DISPLAY_01].Layout[3].wgt > 800 THEN
		OPCuA_Display[CONSTANT_DISPLAY_01].Layout[3].cus := 2;
		OPCuA_Display[CONSTANT_DISPLAY_01].Layout[3].prg := 2;
		OPCuA_Display[CONSTANT_DISPLAY_01].Layout[3].cat := 2;
	END_IF

	//LAYOUT 04
	IF OPCuA_Display[CONSTANT_DISPLAY_01].Layout[4].wgt > 900 THEN
		OPCuA_Display[CONSTANT_DISPLAY_01].Layout[4].wgt := 0;
	END_IF

	IF OPCuA_Display[CONSTANT_DISPLAY_01].Layout[4].wgt > 400 THEN
		OPCuA_Display[CONSTANT_DISPLAY_01].Layout[4].displayID := '0';
		OPCuA_Display[CONSTANT_DISPLAY_01].Layout[4].cus := 2;
		OPCuA_Display[CONSTANT_DISPLAY_01].Layout[4].prg := 2;
		OPCuA_Display[CONSTANT_DISPLAY_01].Layout[4].cat := 2;
	END_IF

	IF OPCuA_Display[CONSTANT_DISPLAY_01].Layout[4].wgt > 800 THEN
		OPCuA_Display[CONSTANT_DISPLAY_01].Layout[4].cus := 1;
		OPCuA_Display[CONSTANT_DISPLAY_01].Layout[4].prg := 1;
		OPCuA_Display[CONSTANT_DISPLAY_01].Layout[4].cat := 1;
	END_IF

// DISPLAY 2 *****************************************************************************

	OPCuA_Display[CONSTANT_DISPLAY_02].Layout[1].backcolour := 16#BADA55;

	OPCuA_Display[CONSTANT_DISPLAY_02].Layout[1].displayID := '2';

	OPCuA_Display[CONSTANT_DISPLAY_02].Layout[1].wgt     := OPCuA_Display[CONSTANT_DISPLAY_02].Layout[1].wgt + 2;

	// Layput 01
	IF OPCuA_Display[CONSTANT_DISPLAY_02].Layout[1].wgt > 900 THEN
		OPCuA_Display[CONSTANT_DISPLAY_02].Layout[1].wgt := 0;
	END_IF

	IF OPCuA_Display[CONSTANT_DISPLAY_02].Layout[1].wgt > 400 THEN
		OPCuA_Display[CONSTANT_DISPLAY_02].Layout[1].displayID := '1';
		OPCuA_Display[CONSTANT_DISPLAY_02].Layout[1].cus := 1;
		OPCuA_Display[CONSTANT_DISPLAY_02].Layout[1].prg := 1;
		OPCuA_Display[CONSTANT_DISPLAY_02].Layout[1].cat := 1;
	END_IF

	IF OPCuA_Display[CONSTANT_DISPLAY_02].Layout[1].wgt > 800 THEN
		OPCuA_Display[CONSTANT_DISPLAY_02].Layout[1].cus := 2;
		OPCuA_Display[CONSTANT_DISPLAY_02].Layout[1].prg := 2;
		OPCuA_Display[CONSTANT_DISPLAY_02].Layout[1].cat := 2;
	END_IF

	// DISPLAY 3 *****************************************************************************

	OPCuA_Display[3].Layout[1].backcolour := 16#BADA55;

	OPCuA_Display[3].Layout[1].displayID := '0';

	OPCuA_Display[3].Layout[1].wgt     := OPCuA_Display[3].Layout[1].wgt + 3;

	// Layput 01
	IF OPCuA_Display[3].Layout[1].wgt > 900 THEN
		OPCuA_Display[3].Layout[1].wgt := 0;
	END_IF

	IF OPCuA_Display[3].Layout[1].wgt > 400 THEN
		OPCuA_Display[3].Layout[1].displayID := '3';
		OPCuA_Display[3].Layout[1].cus := 1;
		OPCuA_Display[3].Layout[1].prg := 1;
		OPCuA_Display[3].Layout[1].cat := 1;
	END_IF

	IF OPCuA_Display[3].Layout[1].wgt > 800 THEN
		OPCuA_Display[3].Layout[1].cus := 2;
		OPCuA_Display[3].Layout[1].prg := 2;
		OPCuA_Display[3].Layout[1].cat := 2;
	END_IF

// DISPLAY 4 *****************************************************************************

	OPCuA_Display[4].Layout[1].backcolour := 16#BADA55;

	OPCuA_Display[4].Layout[1].displayID := '0';

	OPCuA_Display[4].Layout[1].wgt     := OPCuA_Display[4].Layout[1].wgt + 4;

	// Layput 01
	IF OPCuA_Display[4].Layout[1].wgt > 900 THEN
		OPCuA_Display[4].Layout[1].wgt := 0;
	END_IF

	IF OPCuA_Display[4].Layout[1].wgt > 400 THEN
		OPCuA_Display[4].Layout[1].displayID := '4';
		OPCuA_Display[4].Layout[1].cus := 1;
		OPCuA_Display[4].Layout[1].prg := 1;
		OPCuA_Display[4].Layout[1].cat := 1;
	END_IF

	IF OPCuA_Display[4].Layout[1].wgt > 800 THEN
		OPCuA_Display[4].Layout[1].cus := 2;
		OPCuA_Display[4].Layout[1].prg := 2;
		OPCuA_Display[4].Layout[1].cat := 2;
	END_IF

	// DISPLAY 5 *****************************************************************************

	OPCuA_Display[5].Layout[1].backcolour := 16#BADA55;

	OPCuA_Display[5].Layout[1].displayID := '0';

	OPCuA_Display[5].Layout[1].wgt     := OPCuA_Display[5].Layout[1].wgt + 5;

	// Layput 01
	IF OPCuA_Display[5].Layout[1].wgt > 900 THEN
		OPCuA_Display[5].Layout[1].wgt := 0;
	END_IF

	IF OPCuA_Display[5].Layout[1].wgt > 400 THEN
		OPCuA_Display[5].Layout[1].displayID := '5';
		OPCuA_Display[5].Layout[1].cus := 1;
		OPCuA_Display[5].Layout[1].prg := 1;
		OPCuA_Display[5].Layout[1].cat := 1;
	END_IF

	IF OPCuA_Display[5].Layout[1].wgt > 800 THEN
		OPCuA_Display[5].Layout[1].cus := 2;
		OPCuA_Display[5].Layout[1].prg := 2;
		OPCuA_Display[5].Layout[1].cat := 2;
	END_IF

	// DISPLAY 6 *****************************************************************************

	OPCuA_Display[6].Layout[1].backcolour := 16#BADA55;

	OPCuA_Display[6].Layout[1].displayID := '0';

	OPCuA_Display[6].Layout[1].wgt     := OPCuA_Display[6].Layout[1].wgt + 6;

	// Layput 01
	IF OPCuA_Display[6].Layout[1].wgt > 900 THEN
		OPCuA_Display[6].Layout[1].wgt := 0;
	END_IF

	IF OPCuA_Display[6].Layout[1].wgt > 400 THEN
		OPCuA_Display[6].Layout[1].displayID := '5';
		OPCuA_Display[6].Layout[1].cus := 1;
		OPCuA_Display[6].Layout[1].prg := 1;
		OPCuA_Display[6].Layout[1].cat := 1;
	END_IF

	IF OPCuA_Display[6].Layout[1].wgt > 800 THEN
		OPCuA_Display[6].Layout[1].cus := 2;
		OPCuA_Display[6].Layout[1].prg := 2;
		OPCuA_Display[6].Layout[1].cat := 2;
	END_IF

END_PROGRAM
```

### Program Logical/OPCuA/OPCuA_BagEncode (IEC)

#### Cyclic.st - Cyclic code
```iecst
PROGRAM _INIT

//	//Copy Address to local vars and single time copy bag into reduce plc load from 5.4#% to 2.68%
	FOR n := 0 TO MAX_BAGS DO
		pOPCuA_Data[n] := ADR(OPCuA_Bag[n].data[0]);
		pBagData[n] := ADR(Bag[n]);
		memcpy(ADR(OPCuA_Bag[n].data[32]),ADR(n),2);
	END_FOR;
	dataSize := SIZEOF(Bag[0]);
END_PROGRAM
PROGRAM _CYCLIC
FOR n := 0 TO MAX_BAGS DO
//FUB uses 16.9% CPU
//	bagEncode.enable := 1;
//	bagEncode.bagIndex := n;
//	bagEncode.bag := Bag[n];
//	bagEncode.pOutputData := ADR(OPCuA_Bag[n].data[0]);
//	bagEncode.outputDataSize := SIZEOF(OPCuA_Bag[n].data);
//	bagEncode();

//Single Memcpy = 3.56% CPU usage with ADR function...
//With single memcpy we have no hard control over byte position so we must so Bag in the correct format..
//															BYTE
//		Prg : USINT; (*Program*)							0
//		Dst : USINT; (*Destination - Only Supertrack*)		1
//		Wgt : UINT; (*Weight*)								2..3
//		Cnt : UINT; (*Count (Items)*)						4..5
//		Ur1 : UINT; (*User 1*)								6..7
//		Bid : UDINT; (*Bag ID - Supertrack ID*)				8..11
//		Cat : UDINT; (*Category*)							12..15
//		Mis : UDINT; (*Batch ID - MIS Mis Server*)			16..19
//		Cus : UDINT; (*Customer *)							20..23
//		Ur2 : UDINT; (*User 2*)								24..27
//		Timestamp : DATE_AND_TIME;							28..31
//		Bag Index;	UNIT									32..33
		memcpy(pOPCuA_Data[n],pBagData[n],dataSize);

END_FOR;

END_PROGRAM
```

#### Variables.var - Local variables
```iecst
VAR
	n : INT;
	bagString : STRING[150];
	myValue : STRING[30];
	bagEncode : OPCuA_BagEncode_Bin;
	test : UDINT;
	testData : ARRAY[0..33] OF USINT;
	pOPCuA_Data : ARRAY[0..MAX_BAGS] OF UDINT;
	dataSize : UDINT;
	pBagData : ARRAY[0..MAX_BAGS] OF UDINT;
END_VAR
```

### Program Logical/OPCuA/OPCuA_Displays (IEC, version 1.01.0)

#### Cyclic.st - Cyclic code
```iecst
(********************************************************************
 * COPYRIGHT -- Kannegiesser UK
 ********************************************************************
 * PROGRAM: Display
 * File: Display.st
 * Author: T.Reamsbottom
 * Created: Feb 24, 2016
 ********************************************************************
 * Implementation OF PROGRAM Display
 ********************************************************************)
//V1.00.1 First Release.

PROGRAM _INIT
	//Set Default values
	backcolour := 16#0008;
	index := 1;
	FOR n := 1 TO MAX_DISPLAYS DO
		//Set the display and layout vars...
		FOR i := 1 TO 1 DO
			display[n].Layout[i].bag := 220 + index;
			//Set station name as String
			stnIndex := UINT_TO_STRING(index);
			stnName := CONCAT('ES',stnIndex);

			display[n].Layout[i].displayID := stnName;//Only set if required.
			display[n].Layout[i].backcolour := 0;// only set if a custom backcolour is required.
			index := index + 1;
		END_FOR;
	END_FOR;
	// Get size of bag to redure load on PLC
	sizeBag := SIZEOF(Bag[0]);
END_PROGRAM

PROGRAM _CYCLIC

	FOR n:= 1 TO MAX_DISPLAYS DO
		FOR i := 1 TO MAX_LAYOUTS DO
			//Reference to simple Var.
			layout ACCESS ADR(display[n].Layout[i]);
			//Check if data has been set by OPCuA Client
			IF (OPCuA_Display[n].Layout[i].data[43] = 1) THEN
				decodeDisplay.enable := 1;
				decodeDisplay.pInputData := ADR(OPCuA_Display[n].Layout[i].data);
				decodeDisplay.pBag := ADR(Bag[layout.bag]);
				decodeDisplay.sizeBag := sizeBag;
				decodeDisplay();
				IF decodeDisplay.status = ERR_OK THEN // When decode is complete, set write bit to 0
					OPCuA_Display[n].Layout[i].data[43] := 0;
				END_IF;
			ELSIF (OPCuA_Display[n].Layout[i].data[43] = 2) THEN
				memset(ADR(OPCuA_Display[n].Layout[i]),50,SIZEOF(OPCuA_Display[n].Layout[i]));
				OPCuA_Display[n].Layout[i].data[43] := 3;
			ELSIF (OPCuA_Display[n].Layout[i].data[43] >= 2) THEN
				OPCuA_Display[n].Layout[i].data[43] := OPCuA_Display[n].Layout[i].data[43] + 1;
				IF (OPCuA_Display[n].Layout[i].data[43] >= 100) THEN
					OPCuA_Display[n].Layout[i].data[43] := 0;
				END_IF;
			ELSE // Send data
				//Set Default Back colour
				IF layout.backcolour = 0 THEN
					layout.backcolour := backcolour;
				END_IF;
				//Bag Data
				layout.bagData := Bag[layout.bag];
				IF (UINT_TO_INT(layout.bagData.Wgt) < 0) THEN
					layout.bagData.Wgt := 0;
				END_IF;
				//Encode the data to binary for more efficient OPC Comms.

				encodeDisplay.enable := 1;
				encodeDisplay.displayIndex := n;
				encodeDisplay.layoutIndex := i;
				encodeDisplay.layoutData := layout;
				encodeDisplay();
				IF encodeDisplay.status = ERR_OK THEN
					memcpy(ADR(OPCuA_Display[n].Layout[i]),ADR(encodeDisplay.outputData),SIZEOF(OPCuA_Display[n].Layout[i]));
				END_IF;
			END_IF;
		END_FOR;//Layout
	END_FOR;//Display

END_PROGRAM
```

#### Variables.var - Local variables
```iecst
VAR
	display : ARRAY[0..MAX_DISPLAYS] OF Display_typ;
	n : UINT;
	i : UINT;
	layout : REFERENCE TO DispLayout_typ;
	backcolour : UINT;
	stnName : STRING[5];
	stnIndex : STRING[5];
	index : UINT;
	encodeDisplay : OPCuA_DisplayEncode_Bin;
	decodeDisplay : OPCuA_DisplayDecode;
	testTim : BOOL;
	sizeBag : UDINT;
END_VAR
```

### Library Logical/OPCuA/OPCuA (IEC)

#### Constants.var
```iecst
(*Constants*)
VAR CONSTANT
	MAX_DISPLAYS : USINT := 8; (*Maximum number of displays*)
	MAX_LAYOUTS : USINT := 9; (*Maximum number of layouts per display*)
END_VAR
```

#### OPCuA.typ
```iecst
TYPE
	OPCuA_Display_typ : 	STRUCT
		Layout : ARRAY[0..MAX_LAYOUTS]OF DisplayLayoutEncoded_Typ;
	END_STRUCT;
	DispLayout_typ : 	STRUCT
		bag : UINT;
		displayID : STRING[5];
		backcolour : UINT;
		bagData : DispBag_typ;
	END_STRUCT;
	Display_typ : 	STRUCT
		Layout : ARRAY[0..MAX_LAYOUTS]OF DispLayout_typ;
	END_STRUCT;
	DispBag_typ : 	STRUCT  (*//Declare bag twice as the libary does not have access to global vars*)
		Prg : USINT; (*Program*)
		Dst : USINT; (*Destination - Only Supertrack*)
		Wgt : UINT; (*Weight*)
		Cnt : UINT; (*Count (Items)*)
		Ur1 : UINT; (*User 1*)
		Bid : UDINT; (*Bag ID - Supertrack ID*)
		Cat : UDINT; (*Category*)
		Mis : UDINT; (*Batch ID - MIS Mis Server*)
		Cus : UDINT; (*Customer *)
		Ur2 : UDINT; (*User 2*)
		Timestamp : DATE_AND_TIME;
	END_STRUCT;
	DisplayLayoutEncoded_Typ : 	STRUCT
		data : ARRAY[0..43]OF USINT;
	END_STRUCT;
	EncodedBag_typ : 	STRUCT
		data : ARRAY[0..33]OF USINT;
	END_STRUCT;
END_TYPE
```

#### OPCuA.fun - Exported functions and function blocks
```iecst
FUNCTION_BLOCK OPCuA_DisplayEncode_Bin (*TODO: Add your comment here*) (*$GROUP=User,$CAT=User,$GROUPICON=User.png,$CATICON=User.png*)
	VAR_INPUT
		enable : BOOL;
		displayIndex : UINT;
		layoutIndex : UINT;
		layoutData : DispLayout_typ;
	END_VAR
	VAR_OUTPUT
		status : UINT;
		outputData : ARRAY[0..43] OF USINT;
	END_VAR
END_FUNCTION_BLOCK

FUNCTION_BLOCK OPCuA_DisplayEncode_String
	VAR_INPUT
		enable : BOOL;
		displayIndex : UINT;
		layoutIndex : UINT;
		layoutData : DispLayout_typ;
	END_VAR
	VAR_OUTPUT
		status : UINT;
		outputString : STRING[110];
	END_VAR
	VAR
		buildString : STRING[110];
		myValue : STRING[16];
	END_VAR
END_FUNCTION_BLOCK

FUNCTION_BLOCK OPCuA_BagEncode_Bin (*Encode Bag data in USINT For OPCuA comms*) (*$GROUP=User,$CAT=User,$GROUPICON=User.png,$CATICON=User.png*)
	VAR_INPUT
		enable : BOOL;
		bagIndex : UINT;
		bag : DispBag_typ;
		pOutputData : UDINT; (*pointer to output data*)
		outputDataSize : UDINT; (*sixe of output data*)
	END_VAR
	VAR_OUTPUT
		status : UINT;
		outputData : ARRAY[0..33] OF USINT;
	END_VAR
	VAR
		buildData : REFERENCE TO ARRAY[0..33] OF USINT;
	END_VAR
END_FUNCTION_BLOCK

FUNCTION_BLOCK OPCuA_DisplayDecode (**Decode the OPCuA vars into display type.*) (*$GROUP=User,$CAT=User,$GROUPICON=User.png,$CATICON=User.png*)
	VAR_INPUT
		enable : BOOL;
		pInputData : {REDUND_UNREPLICABLE} UDINT; (**pointer to input data*)
		pBag : {REDUND_UNREPLICABLE} UDINT; (**pointer to bag data*)
		sizeBag : UDINT; (**size of Bag structure*)
	END_VAR
	VAR_OUTPUT
		status : UINT;
	END_VAR
END_FUNCTION_BLOCK
```

#### OPCuA_DisplayEncodeString.st
```iecst
(* TODO: Add your comment here *)
FUNCTION_BLOCK OPCuA_DisplayEncode_String
	IF enable THEN
		status := ERR_FUB_BUSY;

		//Build String
		buildString := '';
		//Start with Bag Index.
		itoa(displayIndex,ADR(myValue));
		buildString := myValue;
		buildString := CONCAT(buildString,';');

		itoa(layoutIndex,ADR(myValue));
		buildString := CONCAT(buildString,myValue);
		buildString := CONCAT(buildString,';');

		itoa(layoutData.bagData.Prg,ADR(myValue));
		buildString := CONCAT(buildString,myValue);
		buildString := CONCAT(buildString,';');

		itoa(layoutData.bagData.Cat,ADR(myValue));
		buildString := CONCAT(buildString,myValue);
		buildString := CONCAT(buildString,';');

		itoa(layoutData.bagData.Cus,ADR(myValue));
		buildString := CONCAT(buildString,myValue);
		buildString := CONCAT(buildString,';');

		itoa(layoutData.bagData.Wgt,ADR(myValue));
		buildString := CONCAT(buildString,myValue);
		buildString := CONCAT(buildString,';');

		itoa(layoutData.bagData.Cnt,ADR(myValue));
		buildString := CONCAT(buildString,myValue);
		buildString := CONCAT(buildString,';');

		itoa(layoutData.bagData.Mis,ADR(myValue));
		buildString := CONCAT(buildString,myValue);
		buildString := CONCAT(buildString,';');

		itoa(layoutData.bagData.Ur1,ADR(myValue));
		buildString := CONCAT(buildString,myValue);
		buildString := CONCAT(buildString,';');

		itoa(layoutData.bagData.Ur2,ADR(myValue));
		buildString := CONCAT(buildString,myValue);
		buildString := CONCAT(buildString,';');

		buildString := CONCAT(buildString,layoutData.displayID);
		buildString := CONCAT(buildString,';');

		itoa(layoutData.backcolour,ADR(myValue));
		buildString := CONCAT(buildString,myValue);

		outputString := buildString;
		status := ERR_OK;
	ELSE
		status := ERR_FUB_ENABLE_FALSE;
	END_IF;
END_FUNCTION_BLOCK
```

#### OPCuA_DisplayEncode_Bin.st
```iecst
(* TODO: Add your comment here *)
FUNCTION_BLOCK OPCuA_DisplayEncode_Bin
	IF enable THEN
		status := ERR_FUB_BUSY;
		//Copy Bag data...
		memcpy(ADR(outputData[0]),ADR(layoutData.bagData),SIZEOF(layoutData.bagData));
		//display ID STRING[5] 5 bytes
		memcpy(ADR(outputData[32]),ADR(layoutData.displayID),5);
		//display back Colour
		memcpy(ADR(outputData[37]),ADR(layoutData.backcolour),2);
		//Display Index Index.
		memcpy(ADR(outputData[39]),ADR(displayIndex),2);
		//Index Layout 2 bytes
		memcpy(ADR(outputData[41]),ADR(layoutIndex),2);
		//Clien Write...
		outputData[43] := 0;
		status := ERR_OK;
	ELSE
		status := ERR_FUB_ENABLE_FALSE;
	END_IF;
END_FUNCTION_BLOCK
```

#### OPCuA_BagEncode_Bin.st
```iecst
(* Encode Bag data in USINT For OPCuA comms *)
FUNCTION_BLOCK OPCuA_BagEncode_Bin
	IF enable THEN
		status := ERR_FUB_BUSY;

		//Clear old data,
		buildData ACCESS pOutputData;
		IF outputDataSize >= SIZEOF(buildData) THEN
			//Start with display Index Index.
			memcpy(ADR(buildData[0]),ADR(bagIndex),2);
			//Bag program USINT 1 Byte
			memcpy(ADR(buildData[2]),ADR(bag.Prg),1);
			//Bag destination USINT 1 Byte
			memcpy(ADR(buildData[3]),ADR(bag.Dst),1);
			//Bag Weight UINT 2 bytes
			memcpy(ADR(buildData[4]),ADR(bag.Wgt),2);
			//Bag Count UINT 2 bytes
			memcpy(ADR(buildData[6]),ADR(bag.Cnt),2);
			//Bag UR1 UINT 2 bytes
			memcpy(ADR(buildData[8]),ADR(bag.Ur1),2);
			//Bag bid UDINT 4 bytes
			memcpy(ADR(buildData[10]),ADR(bag.Ur1),4);
			//Bag Category UDINT 4 bytes
			memcpy(ADR(buildData[14]),ADR(bag.Cat),4);
			//Bag Customer UDINT 4 bytes
			memcpy(ADR(buildData[18]),ADR(bag.Cus),4);
			//Bag UR2 UDINT 4 bytes
			memcpy(ADR(buildData[22]),ADR(bag.Ur2),4);
			//Bag Timestamp DATE_AND_TIME 4 bytes
			memcpy(ADR(buildData[26]),ADR(bag.Timestamp),4);
			//Bag Batch ID UDINT (May expand to GUID)
			memcpy(ADR(buildData[30]),ADR(bag.Mis),4);

			status := ERR_OK;
		ELSE
			status := 35624;
		END_IF;
	ELSE
		status := ERR_FUB_ENABLE_FALSE;
	END_IF;

END_FUNCTION_BLOCK
```

#### OPCuA_DisplayDecode.st
```iecst
(* *Decode the OPCuA vars into display type. *)
FUNCTION_BLOCK OPCuA_DisplayDecode
	IF enable THEN
		status := ERR_FUB_BUSY;
		memcpy(pBag,pInputData,sizeBag);
		status := ERR_OK;
	ELSE
		status := ERR_FUB_ENABLE_FALSE;
	END_IF;

END_FUNCTION_BLOCK
```

### PSU.var
```iecst
VAR
	PSU : ARRAY[0..MAX_PSU] OF psu_typ;
END_VAR
(*Constants*)
VAR CONSTANT
	MAX_CHANNELS : USINT := 8;
	PSU_ALM_INDEX : USINT := 20; (*Index alarm text starts at for PSU errors*)
	MAX_PSU : USINT := 2;
END_VAR
```

### PSU.typ
```iecst
TYPE
	psu_typ : 	STRUCT
		Status : psu_channel_typ;
		Fault : psu_channel_typ;
		ton_channelStatus : ARRAY[0..MAX_CHANNELS]OF TON_10ms;
	END_STRUCT;
	psu_channel_typ : 	STRUCT
		channel : ARRAY[0..8]OF BOOL;
	END_STRUCT;
END_TYPE
```

### Program Logical/BlockPSU/zzBlockPSU (IEC)

#### Main.st - Init, cyclic, exit code
```iecst
//Interface Manager to work with BLOCK Electronic Fuse
//Works on a pulse signal basis with 17 bits... Must be called cylically at 10ms.. Ignore rate in documentation, Run at max 200ms pulse.
//V1.00 - First Release
PROGRAM _INIT
scanCount[x] := 1;
step[x] := 0;
refreshTime := 500;//5 second cycle to read data
init[x] := 1;
END_PROGRAM

PROGRAM _CYCLIC
i_readBit[1] := X[2].X01;//Input to read data pulses
i_readBit[2] := X[2].X02;
useExtendedComms := 0;//Use 17 or 89 bit comms.

FOR x := 1 TO MAX_PSU DO

	o_sendBit[x] := 0;

	//Regulate Scan Count to ensure pulse on step[x], and regulate to 70ms Scan time.
	scanCount[x] := scanCount[x] + 1;
	//Create Pulse step[x]s..
	IF (scanCount[x] > 20) THEN
		IF step[x] < 17 THEN
			step[x] := step[x] + 1;
		END_IF;
		scanCount[x] := 1;
	END_IF

	ton_TimeOut[x].IN := (step[x] =17);
	ton_TimeOut[x].PT := 3000;
	ton_TimeOut[x]();

	IF ton_TimeOut[x].Q THEN
		step[x] := 100;
	END_IF;

	o_pulse[x] := (scanCount[x] <= 10);
	ton_reset[x].IN := (step[x] = 99) AND NOT i_readBit[x];
	ton_reset[x].PT := 50;//Minumum time between reading..
	ton_reset[x]();

	ton_refresh[x].IN := (step[x] = 100) AND NOT i_readBit[x];
	ton_refresh[x].PT := refreshTime;
	ton_refresh[x]();

	CASE step[x] OF

		0: //Start Transmission. Set bit to 0

		1..8://1-8 are the required States of the channels
			o_sendBit[x] := 1;
			PSU[x].Status.channel[9-step[x]] := i_readBit[x];
		9: //Use the first 8 bits of this transmission .. (Set to to True to reset[x])
		 	o_sendBit[x] := reset[x];
			PSU[x].Fault.channel[8] := i_readBit[x];
		10://Frame Length;0 = 17 bit,  1=89bit.
			o_sendBit[x] := useExtendedComms;
			PSU[x].Fault.channel[7] := i_readBit[x];
		11://Set values to read//must use extendmode
			o_sendBit[x] := 0;
			PSU[x].Fault.channel[6] := i_readBit[x];
		12..16://Do nothing.
			o_sendBit[x] := 0;
			PSU[x].Fault.channel[17-step[x]] := i_readBit[x];
		17: //Wait for respose from unit.
			o_sendBit[x] := 0;
			o_pulse[x] := useExtendedComms;
			IF i_readBit[x] AND NOT useExtendedComms THEN
				reset[x] := 0;
				step[x] := 99;
			END_IF;
		18..88://Extended data to recieve.
			o_sendBit[x] := 0;
			o_pulse[x] := o_pulse[x] AND useExtendedComms;
		89:
			o_sendBit[x] := 0;
			o_pulse[x] := 0;
			IF i_readBit[x] AND useExtendedComms THEN
				reset[x] := 0;
				step[x] := 99;
			END_IF;
		99://Ack and restart cycle.
			o_sendBit[x] := 0;
			o_pulse[x] := 0;
			//reset[x] cycle. Must wait minimum 200ms
			IF ton_reset[x].Q THEN
				step[x] := 100;
			END_IF;
		100://Idle...
			o_sendBit[x] := 0;
			o_pulse[x] := 0;
			init[x] := 0;

			//Wait to check status 30 sec cycle..
			IF ton_refresh[x].Q OR reset[x] THEN
				step[x] := 0;
				scanCount[x] := 1;
			END_IF;

	END_CASE;

//Ensure Pulse is generated. Always set output to
Y[2].Y01	:= (o_sendBit[1] AND NOT o_pulse[1]) OR (o_pulse[1] AND NOT o_sendBit[1]);
Y[2].Y02	:= (o_sendBit[2] AND NOT o_pulse[2]) OR (o_pulse[2] AND NOT o_sendBit[2]);
//Alarms
	//reset[x] := 0;
	FOR n:= 1 TO MAX_CHANNELS DO
		PSU[x].ton_channelStatus[n].IN := NOT PSU[x].Status.channel[n] AND NOT init[x];
		PSU[x].ton_channelStatus[n].PT := 50;
		PSU[x].ton_channelStatus[n]();

		//Alarm.Active[PSU[x]_ALM_INDEX + n] := ton_channelStatus[n].Q;
		//IF Alarm.Acknowledged[PSU[x]_ALM_INDEX + n] THEN
		//	reset[x] := 1;
		//END_IF;
	END_FOR; //CHANNEL LOOP
END_FOR;//PSU LOOP

END_PROGRAM
```

#### Variables.var - Local variables
```iecst
VAR
	step : ARRAY[0..MAX_PSU] OF UINT;
	i_readBit : ARRAY[0..MAX_PSU] OF BOOL;
	o_sendBit : ARRAY[0..MAX_PSU] OF BOOL;
	scanCount : ARRAY[0..MAX_PSU] OF UINT;
	reset : {REDUND_UNREPLICABLE} ARRAY[0..MAX_PSU] OF BOOL;
	useExtendedComms : BOOL;
	o_pulse : ARRAY[0..MAX_PSU] OF BOOL;
	ton_reset : ARRAY[0..MAX_PSU] OF TON_10ms;
	ton_refresh : ARRAY[0..MAX_PSU] OF TON_10ms;
	refreshTime : UDINT;
	n : USINT;
	init : ARRAY[0..MAX_PSU] OF BOOL;
	ton_TimeOut : ARRAY[0..MAX_PSU] OF TON_10ms;
	x : UINT;
END_VAR
```

### Notes.txt
```
V1.00 First version
	Only tested with 17bit comm. Functionality is questionable as only i need the output wired to the IO circuit for comms.
	?? Should we use addition DM, with PLC main supply for this comms?
```

### CustomLogs.typ - Global data types
```iecst
(********************************************************************
 * COPYRIGHT -- HP
 ********************************************************************
 * Package: CustomLogs
 * File: CustomLogs.typ
 * Author: treamsbottom
 * Created: November 06, 2014
 ********************************************************************
 * Data types of package CustomLogs
 ********************************************************************)

TYPE
	LoggerModule_typ : 	STRUCT
		ident : UDINT;
		len : UDINT;
		memType : UDINT;
		ActIndex : UDINT;
		FormatVer : UDINT;
	END_STRUCT;
	Log_typ : 	STRUCT
		ErrorNo : UDINT;
		Level : UDINT;
		pBinaryData : UDINT;
		lenBinaryData : UDINT;
		pAsciiString : UDINT;
	END_STRUCT;
END_TYPE
```

### CustomLogs.var - Global variables
```iecst
(********************************************************************
 * COPYRIGHT -- HP
 ********************************************************************
 * Package: CustomLogs
 * File: CustomLogs.var
 * Author: treamsbottom
 * Created: November 06, 2014
 ********************************************************************
 * Variables of package CustomLogs
 ********************************************************************)
VAR CONSTANT
	dec_C_MaxCustomLogs : UINT := 400;
END_VAR
VAR
	CustomLog : ARRAY[0..dec_C_MaxCustomLogs] OF Log_typ := [100(0)];
END_VAR
```

### Program Logical/CustomLogs/zzWeighLog (IEC) - *DO NOT USE

#### zzWeighLog.ab - Implementation code
```automation-basic
(* COPYRIGHT -- HP
********************************************************************
* PROGRAM: zzLogger
* File: zzLogger.ab
* Author: treamsbottom
* Created: November 06, 2014
********************************************************************
* Implementation OF PROGRAM zzLogger
	********************************************************************)
PROGRAM _INIT
	pLoggerName = ADR("Weigh") ; Name of Logger module
END_PROGRAM

PROGRAM _CYCLIC

	LOOP n = 0 TO MAX_WEIGH_LOGS DO
		ftrig_OK[n].CLK = StnOK[n]
		ftrig_OK[n] FUB F_TRIG()
		IF ftrig_OK[n].Q AND (weighLog[n].ErrorNo = 0) THEN
			itoa(n,ADR(modNumString))
			strcpy(ADR(errorString[n]),ADR("WeighModule Failed - "))
			strcat(ADR(errorString[n]),ADR(modNumString))
			weighLog[n].ErrorNo = 400
			weighLog[n].Level = arlogLEVEL_WARNING
			weighLog[n].pAsciiString = ADR(errorString[n])
			weighLog[n].lenBinaryData = SIZEOF(X[n])
			weighLog[n].pBinaryData = ADR(X[n])
			shuffle = TRUE
		ENDIF
	ENDLOOP

	;Shuffle Logs...
	//IF shuffle THEN
	LOOP n = 0 TO (dec_C_MaxCustomLogs - 1) DO
		IF (weighLog[n + 1].ErrorNo > 0) AND (weighLog[n].ErrorNo = 0) THEN
			weighLog[n] = weighLog[n + 1]
			weighLog[n + 1] = EmptyLog
		ENDIF
	ENDLOOP
	//ENDIF

	;Write log to logger..
	CASE CustomLogger OF

		ACTION e0_Idle:
			LocalLog = weighLog[0]
			IF (LocalLog.ErrorNo > 0) THEN
				CustomLogger = e1_CheckIfLogExists
			ENDIF
		ENDACTION

		ACTION e1_CheckIfLogExists:
			GetLogInfo.enable = TRUE
			GetLogInfo.pName = pLoggerName
			GetLogInfo FUB AsArLogGetInfo()
			IF GetLogInfo.status = ERR_OK THEN
				LoggerModule.ident = GetLogInfo.ident
				LoggerModule.len = GetLogInfo.len
				LoggerModule.memType = GetLogInfo.memType
				LoggerModule.ActIndex = GetLogInfo.actualIndex
				LoggerModule.FormatVer = GetLogInfo.FormatVer
				CustomLogger = e3_WriteLog
			ELSE IF GetLogInfo.status = arlogERR_NOTEXISTING THEN
				CustomLogger = e2_CreateLog
			ENDIF
		ENDACTION

		ACTION e2_CreateLog:
			CreateLog.enable = TRUE
			CreateLog.pName = pLoggerName
			CreateLog.len = 204800
			CreateLog.memType = arlogUSRROM
			CreateLog FUB AsArLogCreate()
			IF CreateLog.status = ERR_OK THEN
				CustomLogger = e1_CheckIfLogExists
			ENDIF
		ENDACTION

		ACTION e3_WriteLog:

			WriteLog.enable = (LoggerModule.ident > 0)
			WriteLog.ident = LoggerModule.ident
			WriteLog.logLevel = LocalLog.Level
			WriteLog.errornr = LocalLog.ErrorNo
			WriteLog.mem = LocalLog.pBinaryData
			WriteLog.len = LocalLog.lenBinaryData
			WriteLog.asciiString = LocalLog.pAsciiString
			WriteLog FUB AsArLogWrite()
			IF (WriteLog.status = ERR_OK) THEN
				LocalLog = EmptyLog
				weighLog[0] = EmptyLog
				CustomLogger = e0_Idle
			ELSE IF (LoggerModule.ident	 = 0) THEN
				CustomLogger = e0_Idle
			ELSE IF WriteLog.status = arlogERR_ILL_LOGLEVEL THEN
				LocalLog.Level = arlogLEVEL_INFO
			ENDIF
		ENDACTION

	ENDCASE

END_PROGRAM
```

#### zzWeighLog.var - Local variables
```iecst
(********************************************************************
 * COPYRIGHT -- HP
 ********************************************************************
 * Program: zzLogger
 * File: zzLogger.var
 * Author: treamsbottom
 * Created: November 06, 2014
 ********************************************************************
 * Local variables of program zzLogger
 ********************************************************************)
VAR
	LoggerModule : LoggerModule_typ := (0);
END_VAR
VAR CONSTANT
	MAX_WEIGH_LOGS : UINT := 100;
END_VAR
VAR
	WriteLog : AsArLogWrite;
	LocalLog : Log_typ;
END_VAR
VAR CONSTANT
	EmptyLog : Log_typ := (0);
END_VAR
VAR
	CustomLogger : Logger_enum;
	GetLogInfo : AsArLogGetInfo;
	pLoggerName : UDINT;
	CreateLog : AsArLogCreate;
	n : UINT;
	ftrig_OK : ARRAY[0..dec_C_MaxCustomLogs] OF F_TRIG;
	modNumString : STRING[10];
	errorString : ARRAY[0..400] OF STRING[50];
	shuffle : BOOL;
	ton_debounce : ARRAY[0..400] OF TON_10ms;
	testTim : BOOL;
	weighLog : ARRAY[0..MAX_WEIGH_LOGS] OF Log_typ;
END_VAR
```

### Program Logical/CustomLogs/zzWeighStatus (IEC) - *Write Error messages to log on block failure

#### zzModuleLog.var
```iecst
(********************************************************************
 * COPYRIGHT -- HP
 ********************************************************************
 * Program: zzLogger
 * File: zzLogger.var
 * Author: treamsbottom
 * Created: November 06, 2014
 ********************************************************************
 * Local variables of program zzLogger
 ********************************************************************)
VAR CONSTANT
	MAX_MODULE_LOGS : UINT := 20;
END_VAR
VAR
	ModuleLog : ARRAY[0..MAX_MODULE_LOGS] OF Log_typ;
	WriteLog : AsArLogWrite;
	LocalLog : Log_typ;
	CustomLogger : Logger_enum;
	GetLogInfo : AsArLogGetInfo;
	pLoggerName : UDINT;
	CreateLog : AsArLogCreate;
	n : UINT;
	modNumString : STRING[10];
	errorString : ARRAY[0..MAX_MODULE_LOGS] OF STRING[50];
	shuffle : BOOL;
	testTim : BOOL;
	binaryData : ARRAY[0..15] OF BOOL;
	x : UINT;
	nextPos : UINT;
END_VAR
VAR CONSTANT
	EmptyLog : LoggerModule_typ := (ident:=0,len:=0,memType:=0,ActIndex:=0,FormatVer:=0);
END_VAR
VAR
	comp : DINT;
	lastState : ARRAY[0..MAX_MODULE_LOGS] OF BOOL;
	WeighStatus : ARRAY[0..49] OF USINT;
	LoggerModule : LoggerModule_typ := (0);
END_VAR
```

#### zzModuleLog.ab
```automation-basic
(* COPYRIGHT -- HP
********************************************************************
* PROGRAM: zzModuleLog
* File: zzModuleLog.ab
* Author: treamsbottom
* Created: September 14, 2016
********************************************************************
* Implementation OF PROGRAM zzModuleLog
	********************************************************************)

;** V1.00.1 -- T.R -- First Release.. Logs and module OK fail to logbook.. The IO data is stored.. the first 8bits are X the last 8 bits are Y.
PROGRAM _INIT
	pLoggerName = ADR("W_sta") ; Name of Logger module
END_PROGRAM

PROGRAM _CYCLIC

	//Monitor any changes in OK bits
	comp =	memcmp(ADR(WeighStatus),ADR(lastState),SIZEOF(lastState))

	IF (comp <> 0) THEN // State Change detected... Log for difference and write log
		LOOP n = 0 TO MAX_MODULE_LOGS DO
			IF  (WeighStatus[n] <> lastState[n]) AND (WeighStatus[n] > 0) THEN
				itoa(n,ADR(modNumString))
				strcpy(ADR(errorString[n]),ADR("Weight Error - "))
				strcat(ADR(errorString[n]),ADR(modNumString))
				//Find next log position
				nextPos = 0
				LOOP x = 0 TO MAX_MODULE_LOGS DO
					IF ModuleLog[x].ErrorNo = 0 THEN
						nextPos = x
					ENDIF
					EXITIF 	(nextPos > 0)
				ENDLOOP
				ModuleLog[nextPos].ErrorNo = 402
				ModuleLog[nextPos].Level = arlogLEVEL_WARNING
				ModuleLog[nextPos].pAsciiString = ADR(errorString[n])
				ModuleLog[nextPos].lenBinaryData = SIZEOF(WeighStatus[n])
				ModuleLog[nextPos].pBinaryData = ADR(WeighStatus[n])
			ENDIF
		ENDLOOP
		//Set the last state the same as current state..
		memcpy(ADR(lastState),ADR(WeighStatus),SIZEOF(lastState))
	ENDIF

	;Write log to logger..
	CASE CustomLogger OF

		ACTION e0_Idle:
			LocalLog = ModuleLog[1]
			IF (LocalLog.ErrorNo > 0) THEN
				CustomLogger = e1_CheckIfLogExists
			ENDIF
		ENDACTION

		ACTION e1_CheckIfLogExists:
			GetLogInfo.enable = TRUE
			GetLogInfo.pName = pLoggerName
			GetLogInfo FUB AsArLogGetInfo()
			IF GetLogInfo.status = ERR_OK THEN
				LoggerModule.ident = GetLogInfo.ident
				LoggerModule.len = GetLogInfo.len
				LoggerModule.memType = GetLogInfo.memType
				LoggerModule.ActIndex = GetLogInfo.actualIndex
				LoggerModule.FormatVer = GetLogInfo.FormatVer
				CustomLogger = e3_WriteLog
			ELSE IF GetLogInfo.status = arlogERR_NOTEXISTING THEN
				CustomLogger = e2_CreateLog
			ENDIF
		ENDACTION

		ACTION e2_CreateLog:
			CreateLog.enable = TRUE
			CreateLog.pName = pLoggerName
			CreateLog.len = 204800
			CreateLog.memType = arlogUSRROM
			CreateLog FUB AsArLogCreate()
			IF CreateLog.status = ERR_OK THEN
				CustomLogger = e1_CheckIfLogExists
			ENDIF
		ENDACTION

		ACTION e3_WriteLog:

			WriteLog.enable = (LoggerModule.ident > 0)
			WriteLog.ident = LoggerModule.ident
			WriteLog.logLevel = LocalLog.Level
			WriteLog.errornr = LocalLog.ErrorNo
			WriteLog.mem = LocalLog.pBinaryData
			WriteLog.len = LocalLog.lenBinaryData
			WriteLog.asciiString = LocalLog.pAsciiString
			WriteLog FUB AsArLogWrite()
			IF (WriteLog.status = ERR_OK) THEN
				//LocalLog = EmptyLog
				//ModuleLog[0] = EmptyLog
				//Shuffle Logs
				memcpy(ADR(ModuleLog[0]),ADR(ModuleLog[1]),(SIZEOF(ModuleLog[0]) * (MAX_MODULE_LOGS - 1)))
				CustomLogger = e0_Idle
			ELSE IF (LoggerModule.ident	 = 0) THEN
				CustomLogger = e0_Idle
				memcpy(ADR(ModuleLog[0]),ADR(ModuleLog[1]),(SIZEOF(ModuleLog[0]) * (MAX_MODULE_LOGS - 1)))
			ELSE IF WriteLog.status = arlogERR_ILL_LOGLEVEL THEN
				LocalLog.Level = arlogLEVEL_INFO
			ENDIF
		ENDACTION

	ENDCASE

END_PROGRAM
```

### Program Logical/CustomLogs/zzModuleLog (IEC, version 1.00.1) - *Write Error messages to log on block failure

#### zzModuleLog.ab - Implementation code
```automation-basic
(* COPYRIGHT -- HP
********************************************************************
* PROGRAM: zzModuleLog
* File: zzModuleLog.ab
* Author: treamsbottom
* Created: September 14, 2016
********************************************************************
* Implementation OF PROGRAM zzModuleLog
	********************************************************************)
;** V1.00.1 -- T.R -- First Release.. Logs and module OK fail to logbook.. The IO data is stored.. the first 8bits are X the last 8 bits are Y.

PROGRAM _INIT
	pLoggerName = ADR("Mod_Ok") ; Name of Logger module
END_PROGRAM

PROGRAM _CYCLIC
	//Monitor any changes in OK bits
	comp =	memcmp(ADR(OK),ADR(lastState),SIZEOF(lastState))

	IF (comp <> 0) THEN // State Change detected... Log for difference and write log
		LOOP n = 0 TO MAX_MODULE_LOGS DO
			IF NOT OK[n] AND lastState[n] THEN
				itoa(n,ADR(modNumString))
				strcpy(ADR(errorString[n]),ADR("Module Failed - "))
				strcat(ADR(errorString[n]),ADR(modNumString))
				memcpy(ADR(binaryData[0]),ADR(X[n]),SIZEOF(X[n]))
				memcpy(ADR(binaryData[8]),ADR(Y[n]),SIZEOF(Y[n]))
				//Find next log position
				nextPos = 0
				LOOP x = 0 TO MAX_MODULE_LOGS DO
					IF ModuleLog[x].ErrorNo = 0 THEN
						nextPos = x
					ENDIF
				EXITIF 	(nextPos > 0)
				ENDLOOP
				ModuleLog[nextPos].ErrorNo = 400
				ModuleLog[nextPos].Level = arlogLEVEL_WARNING
				ModuleLog[nextPos].pAsciiString = ADR(errorString[n])
				ModuleLog[nextPos].lenBinaryData = SIZEOF(binaryData)
				ModuleLog[nextPos].pBinaryData = ADR(binaryData[0])
			ENDIF
		ENDLOOP
		//Set the last state the same as current state..
		memcpy(ADR(lastState),ADR(OK),SIZEOF(lastState))
	ENDIF

	;Write log to logger..
	CASE CustomLogger OF

		ACTION e0_Idle:
			LocalLog = ModuleLog[1]
			IF (LocalLog.ErrorNo > 0) THEN
				CustomLogger = e1_CheckIfLogExists
			ENDIF
		ENDACTION

		ACTION e1_CheckIfLogExists:
			GetLogInfo.enable = TRUE
			GetLogInfo.pName = pLoggerName
			GetLogInfo FUB AsArLogGetInfo()
			IF GetLogInfo.status = ERR_OK THEN
				LoggerModule.ident = GetLogInfo.ident
				LoggerModule.len = GetLogInfo.len
				LoggerModule.memType = GetLogInfo.memType
				LoggerModule.ActIndex = GetLogInfo.actualIndex
				LoggerModule.FormatVer = GetLogInfo.FormatVer
				CustomLogger = e3_WriteLog
			ELSE IF GetLogInfo.status = arlogERR_NOTEXISTING THEN
				CustomLogger = e2_CreateLog
			ENDIF
		ENDACTION

		ACTION e2_CreateLog:
			CreateLog.enable = TRUE
			CreateLog.pName = pLoggerName
			CreateLog.len = 204800
			CreateLog.memType = arlogUSRROM
			CreateLog FUB AsArLogCreate()
			IF CreateLog.status = ERR_OK THEN
				CustomLogger = e1_CheckIfLogExists
			ENDIF
		ENDACTION

		ACTION e3_WriteLog:

			WriteLog.enable = (LoggerModule.ident > 0)
			WriteLog.ident = LoggerModule.ident
			WriteLog.logLevel = LocalLog.Level
			WriteLog.errornr = LocalLog.ErrorNo
			WriteLog.mem = LocalLog.pBinaryData
			WriteLog.len = LocalLog.lenBinaryData
			WriteLog.asciiString = LocalLog.pAsciiString
			WriteLog FUB AsArLogWrite()
			IF (WriteLog.status = ERR_OK) THEN
				//LocalLog = EmptyLog
				//ModuleLog[0] = EmptyLog
				//Shuffle Logs
				memcpy(ADR(ModuleLog[0]),ADR(ModuleLog[1]),(SIZEOF(ModuleLog[0]) * (MAX_MODULE_LOGS - 1)))
				CustomLogger = e0_Idle
			ELSE IF (LoggerModule.ident	 = 0) THEN
				CustomLogger = e0_Idle
				memcpy(ADR(ModuleLog[0]),ADR(ModuleLog[1]),(SIZEOF(ModuleLog[0]) * (MAX_MODULE_LOGS - 1)))
			ELSE IF WriteLog.status = arlogERR_ILL_LOGLEVEL THEN
				LocalLog.Level = arlogLEVEL_INFO
			ENDIF
		ENDACTION

	ENDCASE

END_PROGRAM
```

#### zzModuleLog.typ - Local data types
```iecst
(********************************************************************
 * COPYRIGHT -- HP
 ********************************************************************
 * Program: zzLogger
 * File: zzLogger.typ
 * Author: treamsbottom
 * Created: November 06, 2014
 ********************************************************************
 * Local data types of program zzLogger
 ********************************************************************)

TYPE
	Logger_enum :
		(
		e0_Idle,
		e1_CheckIfLogExists,
		e2_CreateLog,
		e3_WriteLog
		);
END_TYPE
```

#### zzModuleLog.var - Local variables
```iecst
(********************************************************************
 * COPYRIGHT -- HP
 ********************************************************************
 * Program: zzLogger
 * File: zzLogger.var
 * Author: treamsbottom
 * Created: November 06, 2014
 ********************************************************************
 * Local variables of program zzLogger
 ********************************************************************)
VAR
	LoggerModule : LoggerModule_typ := (0);
END_VAR
VAR CONSTANT
	MAX_MODULE_LOGS : UINT := 399;
END_VAR
VAR
	ModuleLog : ARRAY[0..MAX_MODULE_LOGS] OF Log_typ;
	WriteLog : AsArLogWrite;
	LocalLog : Log_typ;
	CustomLogger : Logger_enum;
	GetLogInfo : AsArLogGetInfo;
	pLoggerName : UDINT;
	CreateLog : AsArLogCreate;
	n : UINT;
	modNumString : STRING[10];
	errorString : ARRAY[0..MAX_MODULE_LOGS] OF STRING[50];
	shuffle : BOOL;
	testTim : BOOL;
	binaryData : ARRAY[0..15] OF BOOL;
	x : UINT;
	nextPos : UINT;
END_VAR
VAR CONSTANT
	EmptyLog : LoggerModule_typ := (ident:=0,len:=0,memType:=0,ActIndex:=0,FormatVer:=0);
END_VAR
VAR
	comp : DINT;
	lastState : ARRAY[0..MAX_MODULE_LOGS] OF BOOL;
END_VAR
```

### Program Logical/CustomLogs/zzModuleLog1 (IEC, version 1.00.1) - *Advanced Module Logger -- Have to Manually set the block order.
